METHOD PRIVATE push : BOOL
VAR_INPUT
  pNewCT : POINTER TO FB_ContainerDefGrid;
END_VAR
// checks
// - valid param
IF pNewCT = 0 THEN LogError('push: invalid pointer'); RETURN; END_IF
// - list full
IF _nAttachedCTs >= nUpperIndexCTList THEN  // list overflow no free element for processing
  LogError('Worker processing list full, ignore new CT');
  Abort(iCT:=pNewCT^, sReason:='attach failed - too many attached');  // abort new CT (no release because not yet attached)
  RETURN;
END_IF
// - only one CT allowed
IF _nAttachedCTs > 0 AND NOT _bSupportParallelCT THEN
  LogError(Msg:='another container already attached -> ignore new (set error)');
  Abort(iCT:=pNewCt^, sReason:='attach failed - no parallel support');  // abort new CT
END_IF

// add to list
_nAttachedCTs := _nAttachedCTs + 1;
_pAttachedCTList[_nAttachedCTs] := pNewCT;
MEMSET(destAddr:=ADR(_stAttachedCTData[_nAttachedCTs]), fillByte:=0, n:=SIZEOF(_stAttachedCTData[1]));  // clear additional data
_pNewAttachedHdlData := ADR(_stAttachedCTData[_nAttachedCTs]);   // select handling data for new attached ct 

// apply head
IF _nAttachedCTs = 1 THEN
  // set HEAD
  _pAttachedCt := _pAttachedCTList[nLowerIndexCTList];  
  _bAttached := TRUE;

  // start callback on HEAD
  StartCT(pCtDefGrid:=_pAttachedCt);
END_IF

push := TRUE;
END_METHOD

(*
  Release CT from Worker.
  :return: TRUE if CT was released, FALSE if no CT was registered 
*)
METHOD Release : BOOL
VAR_INPUT
  iCT              : I_CT;                         (*container at triggered event position*)
END_VAR
VAR
  nIdx             : DINT;
  pCT              : POINTER TO FB_ContainerDefGrid;
END_VAR
// remove CT -----------------------------------------------------
// -- get real instance
pCT := getCtInst(iCT:=iCT);
IF pCT = 0 THEN LogError('Release: could not find ct instance'); RETURN; END_IF

// remove and release CT
IF pull(pRemCT:=pCT, nRemIndex=>nIdx) THEN
  LogLvl(Lvl:=E_LogSeverity.Debug, Msg:=F_Concat4('Release CT[', TO_STRING(nIdx), '] ', pCt^.print(0)));
  Release := TRUE;  
END_IF
END_METHOD

(*
  Container will be released from tracker (destroyed) and not available anymore. 
*)
METHOD remove
VAR_INPUT
	(*container at triggered event position*)
	iCT	: I_CT;
END_VAR
SUPER^();

// nothing done
// We keep in internal WorkerList until work is done. CT will be removed from tracker.
END_METHOD

METHOD PRIVATE setName : BOOL
VAR_INPUT
  sName : STRING;
END_VAR
VAR
  nIdx : INT;
  bDone : BOOL;
END_VAR
IF sName = '' THEN
  // generate worker name
  _name := THIS^.InstanceName;
  WHILE NOT bDone DO
    nIdx := FIND(_name, '.');
    IF nIdx = 0 THEN bDone := TRUE; EXIT; 
    ELSE
      _name := RIGHT(_name,LEN(_name)-nIdx);
    END_IF 
  END_WHILE
ELSE
  _name := sName;  
END_IF
END_METHOD

METHOD PROTECTED StartCT
VAR_INPUT
 pCtDefGrid   : POINTER TO FB_ContainerDefGrid;
END_VAR
(* Override specific implementation in child class *)
END_METHOD

METHOD PROTECTED StopCT
VAR_INPUT
 pCtDefGrid   : POINTER TO FB_ContainerDefGrid;
END_VAR
(* Override specific implementation in child class *)
END_METHOD

METHOD  work
VAR
  i : UDINT;
  pCt : POINTER TO FB_ContainerDefGrid;
END_VAR
// set tracking offset
_nTrackOffset := F_MeterToSubPixel(fPosMeter:=fPosition, fResoSubPx:=_fPrintResolution*_fSubPxResolution);  // [pos domain] save position

//Work only with attached container
IF _nAttachedCTs = 0 THEN RETURN; END_IF

IF _pAttachedCt <> 0 AND_THEN _pAttachedCt^.pCT <> 0 THEN _nHeadCtId := _pAttachedCt^.pCT^.iId;
ELSE                                                      _nHeadCtId := 0; END_IF

FOR i:=nLowerIndexCTList TO nLowerIndexCTList + _nAttachedCTs - 1 DO
  pCt := _pAttachedCTList[i];

  // update CT position
  _stAttachedCTData[i].fPosRelToAttach := getPosRelToAttach(iCT:=pCt^);
  
  // release CT (manually)
  IF _bForceRelease THEN
    _bForceRelease := FALSE;
    pCt^.AbortDeformation(sReason:='Manually realease CT', Src:=_pEcSrc^, bHideLog:=FALSE);
    Release(iCT:=pCt^);

  // security release 
  ELSIF _fCtSecurityReleasePos > 0 AND (ABS(_stAttachedCTData[i].fPosRelToAttach) > _fCtSecurityReleasePos) THEN
    pCt^.AbortDeformation(sReason:=F_Concat2('Security released CT Id=', TO_STRING(pCt^.pCT^.iId)), Src:=_pEcSrc^, bHideLog:=FALSE);
    Release(iCT:=pCt^);
  END_IF

END_FOR
END_METHOD

END_FUNCTION_BLOCK

// ---- POUs/Print/DefGrid/FB_WorkerDefGrid_Deformation.TcPOU
FUNCTION_BLOCK FB_WorkerDefGrid_Deformation EXTENDS FB_WorkerDefGrid
VAR_INPUT
END_VAR
VAR_OUTPUT
END_VAR
VAR
  // references
  _iParamMediator : I_ParamMediator;
  
  //Worker specific configuration
  _nPrintUnitWidth            : UDINT;  // default print unit width [px]  
  _nImageWidthPx              : UDINT;  // size of the image (width)
  _nImageDepthPx              : UDINT;  // size of the image (depth)
  
  // -
  _bNewJob                    : BOOL;   // new job started 

  //Deformation status (per attached CT)
  _nDeformationProcPoints     : ARRAY[nLowerIndexCTList..nUpperIndexCTList] OF UDINT;  // available grid points on ct
  _nDeformationProcCols       : ARRAY[nLowerIndexCTList..nUpperIndexCTList] OF UDINT;  // number of already generated grid columns
  _eDeformStep                : ARRAY[nLowerIndexCTList..nUpperIndexCTList] OF E_DeformationStep;   // status deformation of ct
  _bDeformationError          : ARRAY[nLowerIndexCTList..nUpperIndexCTList] OF BOOL;   // status deformation of ct
  _bDeformationBusy           : ARRAY[nLowerIndexCTList..nUpperIndexCTList] OF BOOL;   // status deformation of ct
  _bDeformationDone           : ARRAY[nLowerIndexCTList..nUpperIndexCTList] OF BOOL;   // status deformation of ct
  _nDeformationErrorId        : ARRAY[nLowerIndexCTList..nUpperIndexCTList] OF UDINT;  // status deformation of ct
  _tDeformationExecutionTime  : ARRAY[nLowerIndexCTList..nUpperIndexCTList] OF TIME;   // status deformation of ct
  _bAborted                   : ARRAY[nLowerIndexCTList..nUpperIndexCTList] OF BOOL;   // status deformation of ct

  // ui
  eDeformTypeUi : E_DeformationType;
END_VAR 

VAR PERSISTENT
  _sDeformationGridSettings  : ST_DefGridSettings := (   // grid definition settings
                                  nGridPitchX:=GVL_Deformation.nC_DefaultGridPitch_X,   // this must match the hw config (in fpga)
                                  nGridPitchY:=GVL_Deformation.nC_DefaultGridPitch_Y,   // this must match the hw config (in fpag)
                                  eDeformationType:=E_DeformationType.NoDeformation
                             );
  _fDistToCam                : LREAL := 0.02;   // distance to cam worker 
END_VAR

METHOD PROTECTED  Attach : BOOL
VAR_INPUT
  iCT              : I_CT;                         (*container at triggered event position*)
END_VAR
VAR
  i : UDINT;
  bDeformErr : BOOL;
  eDeformStep : E_DeformationStep;
END_VAR
(*Please do enable externally in PrintModule
IF getCtInst(iCT:=iCT, pCT=>pCt) = 0 THEN    // get specific container
  RETURN;
END_IF

//-- (auto-) enable / disable worker based on mode (do before parent Attach(), is checked inside)
bWorkerEnable := _sDeformationGridSettings.eDeformationType <> E_DeformationType.NoDeformation 
                     AND SEL(pCt^.eCamMode > E_CameraMode.NoCorrection, FALSE, TRUE);
*)

// -- Attach
IF NOT SUPER^.Attach(iCT:=iCT) THEN
  RETURN;
END_IF

// Additional worker checks
IF _pNewAttached = 0 THEN RETURN; END_IF

// - Additional worker checks
bDeformErr := _pNewAttached^.getDeformationStatus(eDStep=>eDeformStep);   // get latest status 
  
// - deformation started? and no deformation error so far
IF bDeformErr OR eDeformStep < E_DeformationStep.cameraStarted THEN
  Release(iCT:=iCT);  // nothing to do anymore

  // - job is valid?
ELSIF _pNewAttached^.pJob = 0 OR NOT _bJobActive THEN
  _pNewAttached^.AbortDeformation(sReason:='No valid job', Src:=_pEcSrc^, bHideLog:=FALSE);
  Release(iCT:=iCT);
  
// - did camera start?  
(*ELSIF eDeformStep < E_DeformationStep.cameraStarted THEN
  _pNewAttached^.AbortDeformation(sReason:='Prio steps did not start', Src:=_pEcSrc^);
  Release(iCT:=iCT);
*)
  
// - OK attach
ELSE
  // checks
  IF eDeformStep < E_DeformationStep.cameraStarted THEN LogWarning('Sub-optimal timing, camera did not yet start'); END_IF
  // start deformation
  _pNewAttached^.StartDeformation(
    sDefGridSettings:=_sDeformationGridSettings, 
    fStartDeformationPos:=getPosRelToAttach(iCT)/_fSubPxResolution   // [px]
  );
  Attach := TRUE;
END_IF
END_METHOD

METHOD InitWorkerDeformation : BOOL
VAR_INPUT
  nPrintUnitWidth : UDINT;
  iDefGridParamMediator : I_ParamMediator;
END_VAR
VAR
  i : UDINT;
END_VAR
IF NOT bInitialized THEN LogError('Base Worker not initialized! call init() before'); RETURN; END_IF
IF iDefGridParamMediator = 0 THEN bInitialized := FALSE; LogError('Invalid parameter, no valid param mediator'); RETURN; END_IF


// worker specific init
_nPrintUnitWidth := nPrintUnitWidth;
_iParamMediator := iDefGridParamMediator;
_bNewJob := FALSE;

FOR i:=nLowerIndexCTList TO nUpperIndexCTList DO
  _nDeformationProcPoints[i]     := 0;
  _nDeformationProcCols[i]       := 0;
  _eDeformStep[i]                := 0;
  _bDeformationError[i]          := 0;
  _bDeformationBusy[i]           := 0;
  _bDeformationDone[i]           := 0;
  _nDeformationErrorId[i]        := 0;
  _tDeformationExecutionTime[i]  := T#0S;
  _bAborted[i]                   := 0;
END_FOR
END_METHOD

METHOD mJobStart
VAR_INPUT
	sJobDef	: CalmarCompPrint.I_JobDefinition;
END_VAR
VAR
  sCamSettings : ST_CameraGridSettings;
END_VAR
// check and init invalid settings
IF _iParamMediator = 0 THEN LogError('no parameter mediator'); RETURN; END_IF
IF _sDeformationGridSettings.nGridPitchX = 0 THEN _sDeformationGridSettings.nGridPitchX:=GVL_Deformation.nC_DefaultGridPitch_X; LogError(F_Concat2('nGridPitchX not configured, set default=', TO_STRING(GVL_Deformation.nC_DefaultGridPitch_X))); END_IF
IF _sDeformationGridSettings.nGridPitchY = 0 THEN _sDeformationGridSettings.nGridPitchY:=GVL_Deformation.nC_DefaultGridPitch_Y; LogError(F_Concat2('nGridPitchY not configured, set default=', TO_STRING(GVL_Deformation.nC_DefaultGridPitch_Y))); END_IF
IF _nPrintUnitWidth = 0 THEN LogError('_nPrintUnitWidth not configured'); END_IF
IF fPosition = 0 THEN LogError('No valid Worker position: set it to WorkerCamera.fCameraToPrintOffset + 0.05; '); END_IF

// configuration
// calculate deformation  settings
// - save image y-offset (centered)
// - save image size
_nImageWidthPx := DINT_TO_UDINT(F_MeterToSubPixel(fPosMeter:=sJobDef.fImageWidth/1000, fResoSubPx:=_fPrintResolution));
_nImageDepthPx := DINT_TO_UDINT(F_MeterToSubPixel(fPosMeter:=sJobDef.fImageDepth/1000, fResoSubPx:=_fPrintResolution));
_sDeformationGridSettings.nGridImageOffsetY := LIMIT(0, ((_nPrintUnitWidth - _nImageWidthPx)) / 2, (_nPrintUnitWidth));  // TODO: if you can get this value from PUC use the other one to have a consistent image shift value 

// - calc grid size and number of points
(*
  Use image width / depth in px divide by GridPitch in X/Y to do a ceil(always next bigger integer).
  +1 -> Because Grid starts at 0 until the calculated numbers we have one point more [0, 1, 2, 3] = 4 points (not 3) 
*)
IF _sDeformationGridSettings.nGridPitchX > 0 AND _sDeformationGridSettings.nGridPitchY > 0 THEN
  _sDeformationGridSettings.nGridSizeX := F_Ceil(val:=UDINT_TO_LREAL(_nImageDepthPx)/_sDeformationGridSettings.nGridPitchX) + 1;
  _sDeformationGridSettings.nGridSizeY := F_Ceil(val:=UDINT_TO_LREAL(_nImageWidthPx + _sDeformationGridSettings.nGridImageOffsetY)/_sDeformationGridSettings.nGridPitchY) + 1;
END_IF
_sDeformationGridSettings.nGridPoints :=  _sDeformationGridSettings.nGridSizeX * _sDeformationGridSettings.nGridSizeY;

sCamSettings := _iParamMediator.sCameraGridSettings;
_sDeformationGridSettings.eDeformationType := sCamSettings.eDeformationType;   // apply deformation mode (for ui)
eDeformTypeUi := _sDeformationGridSettings.eDeformationType;

_bJobActive := TRUE;
END_METHOD

METHOD  mJobStop
VAR_INPUT
	sStatus	: CalmarCompPrint.I_JobStatus;
END_VAR
_bJobActive := FALSE;
END_METHOD

(*
  Release CT from Worker.
  :return: TRUE if CT was released, FALSE if no CT was registered 
*)
METHOD Release : BOOL
VAR_INPUT
  iCT              : I_CT;                         (*container at triggered event position*)
END_VAR
VAR
  i                : DINT;
  Index            : DINT;
  LowerIndex       : DINT := 1;
  pCt              : POINTER TO FB_ContainerDefGrid;
  eStep            : E_DeformationStep;
END_VAR
IF iCT = 0 OR _nAttachedCTs = 0 THEN RETURN; END_IF

// release from deformation module
IF getCtInst(iCT:=iCT, pCT=>pCt) = 0 THEN LogError('Release: could not find ct instance'); RETURN; END_IF
IF _iParamMediator <> 0 THEN
  pCt^.getDeformationStatus(eDStep => estep);
  IF estep >= E_DeformationStep.createdScriptContainer THEN
    pCt^.StopScript(iCT:=iCT);
    //_pParamMediator^.ReleaseDeformationCT(iCT:=iCT);
  END_IF
END_IF

Release := SUPER^.Release(iCT:=iCT);
END_METHOD

PROPERTY sDeformationGridSettings : ST_DefGridSettings
GET
sDeformationGridSettings := _sDeformationGridSettings;
END_GET
END_PROPERTY

METHOD setupPosition
VAR
  sCamSettings : ST_CameraGridSettings;
END_VAR
IF _pAttachedCt <> 0 THEN RETURN; END_IF    // Update only without attached container

sCamSettings := _iParamMediator.sCameraGridSettings;

// set tracking offset
fPosition := sCamSettings.fDetectToCam + _fDistToCam;
END_METHOD

METHOD  work
VAR
  i : UDINT;
  pCT : POINTER TO FB_ContainerDefGrid;
END_VAR
//-----------------------------------------------------------
SUPER^.work();      // Parent implementation

setupPosition();    // Worker position update

// Work only with attached container (additional work to Base class)
FOR i:=nLowerIndexCTList TO nLowerIndexCTList + _nAttachedCTs - 1 DO
  pCt := _pAttachedCTList[i];
 
  // update deformation handler
  pCT^.UpdateDeformation(fPos:=_stAttachedCTData[i].fPosRelToAttach/_fSubPxResolution);  // pos in [px]
  
  // get status
  _bDeformationError[i] := pCt^.getDeformationStatus(eDStep => _eDeformStep[i], 
                            bBusy => _bDeformationBusy[i],
                            bDone => _bDeformationDone[i],
                            nErrorId => _nDeformationErrorId[i], 
                            tExecutionTime => _tDeformationExecutionTime[i],
                            bAborted => _bAborted[i]);
  _nDeformationProcPoints[i] := pCt^.nAvailableGridPoints;
  _nDeformationProcCols[i]   := pCt^.nAvailableGridCols;
     
  // Release container when all points have been processed or error
  IF _bDeformationDone[i] OR _bDeformationError[i] THEN
    // tag CT with error if deformation had an error
    IF _bDeformationError[i] THEN 
      IF NOT _bAborted[i] THEN
        pCt^.AbortDeformation(sReason:=F_Concat2('WorkerDeformation: ', EC_DefGrid.ecDefGrid_DefGridError.Desc), Src:=_pEcSrc^, bHideLog:=FALSE);
      //not needed ELSE
      //  pCt^.setError(ErrDef:=EC_DefGrid.ecDefGrid_DefGridError, Src:=_pEcSrc^);
      END_IF
    END_IF
    LogLvl(Lvl:=E_LogSeverity.Detail, Msg:=F_Concat4('Done with: CamP=',  TO_STRING(pCT^.nRegisteredCameraPoints), ' GridP=', TO_STRING(pCt^.nAvailableGridPoints)));
    Release(pCt^);
  END_IF
  
END_FOR
END_METHOD

END_FUNCTION_BLOCK

// ---- POUs/Print/DefGrid/FB_PrintOverview.TcPOU
FUNCTION_BLOCK FB_PrintOverview
VAR_INPUT
  fX_m,  fY_m   : LREAL;    // max. x/y position [m]
  nX_px, nY_px  : DINT;     // max. x/y pixel in view
  fPxToMRatio   : LREAL;    // 
  iPrintPosition : I_PrintPosition;
END_VAR

VAR
  // helper
  bInit   : BOOL;
  nCtr    : UDINT;
  nNum    : UDINT;
  
  // config
  _pCTM   : POINTER TO FB_CTManagerDefGrid;
  _pWorkerDefGrid : POINTER TO FB_WorkerDefGrid;
  _fPrintResolution : LREAL;      // [dpi]
  _fSubPixelResolution : LREAL;   // sub pixel resolution
  
  // Container view list
  iCT     : I_CT;
  aCTV    : ARRAY[1..iCPr_MAX_CONTAINER] OF FB_ContainerView;
  // Worker view list
  iWorker : I_Worker;
  aWorkerV: ARRAY[1..nC_MAX_WORKER_VIEWS] OF FB_ViewPositionControl;
  aWorkerFb: ARRAY[1..nC_MAX_WORKER_VIEWS] OF POINTER TO FB_WorkerDefGrid;
  
  // motion and position
  bMovingInd : BOOL;
  fSpeed  : LREAL;
  fbBlink : FB_BLINK;
  t : TIME;
  
  // last container debug
  nGridRowStart : UDINT;  // starting grid colum for Grid debug Visu
  nGridColStart : UDINT;  // starting grid colum for Grid debug Visu
  pLastCT : POINTER TO FB_ContainerDefGrid;   // pointer to last created container
  
  // time
  sCurrentDateTime : STRING;
  
  // view control
  bShowCtDetails : BOOL;
END_VAR
VAR CONSTANT
  nC_MAX_WORKER_VIEWS : UINT := 10;
END_VAR

IF NOT checkConfig() THEN RETURN; END_IF    // check config

// -- show CTs -----------------------
nNum := _pCTM^.nCount;
FOR nCtr := 1 TO nNum DO
  // get CT interface from list
  iCT := _pCTM^.getCT(nIdx:=nCtr);
  IF iCT <> 0 THEN
    // set position
    aCTV[nCtr].setPos(x:=iCT.GetPosRel(iTracker:=_pCTM^.iTracker), y:=0);

    // display
    aCTV[nCtr].bHide := FALSE;
    aCTV[nCtr]( iCT:=iCT, 
                iIdx:=UDINT_TO_UINT(iCT.pCT^.nMemIndex), 
                fPxtoMRatio:=fPxToMRatio, 
                fPosToMFactor := 0.0254 / (_fPrintResolution*_fSubPixelResolution), 
                iTracker:=_pCTM^.iTracker);
  END_IF
END_FOR

FOR nCtr := (nNum+1) TO iCPr_MAX_CONTAINER DO
  aCTV[nCtr].iCT := 0;
  aCTV[nCtr].bHide := TRUE;
END_FOR

// -- show Workers -----------------------
iWorker := _pWorkerDefGrid^.Root;
nCtr := 0;
WHILE iWorker <> 0 DO     // walk through worker chain
  nCtr := nCtr + 1;
  aWorkerFb[nCtr] := iWorker.Inst;  // get fb pointer
  aWorkerV[nCtr].bHide := FALSE;
  aWorkerV[nCtr].setPos(x:=aWorkerFb[nCtr]^.nTrackOffset, y:=0);
  iWorker:=iWorker.Next;
END_WHILE
FOR nCtr := (nCtr+1) TO nC_MAX_WORKER_VIEWS DO
  aWorkerV[nCtr].bHide := TRUE;
END_FOR

// -- show positioning -----------------------
fSpeed := iPrintPosition.getSpeed();
IF LrealIsNaN(x:=fSpeed) THEN
  fSpeed := 0;
END_IF
t := LREAL_TO_TIME(1000-fSpeed*900);
fbBlink(bI_Enable:=SEL(fSpeed > 0, FALSE, TRUE), tI_Time:=t, bO_Out=>bMovingInd);

// -- last container debug detail ------------
IF _pCTM^.nCount > 0 THEN
  iCT := _pCTM^.getCT(1);
  IF iCT <> 0 THEN  pLastCT := _pCTM^.GetContainerInstance(iCT:=iCT); END_IF
END_IF

// -- current time ---------------------------
sCurrentDateTime := F_TimeGetDateTime();

METHOD checkConfig : BOOL
VAR_INPUT
END_VAR
VAR_INST
  _fX_m, _fY_m   : LREAL;
  _nX_px, _nY_px : DINT; 
END_VAR
VAR
  bOK : BOOL;
END_VAR
IF NOT bInit THEN RETURN; END_IF
IF iPrintPosition = 0 THEN RETURN; END_IF

_fPrintResolution := iPrintPosition.fPrintResolution;
_fSubPixelResolution := iPrintPosition.fSubPxResolution;

// changed settings
IF _fX_m <> fX_m OR
          _fY_m <> fY_m OR
          _nX_px <> nX_px OR
          _nY_px <> nY_px THEN
  // save new config
   _fX_m := fX_m;
   _fY_m := fY_m;
   _nX_px := nX_px;
   _nY_px := nY_px;
   config();
END_IF

checkConfig := TRUE;
END_METHOD

METHOD PRIVATE config
VAR_INPUT
END_VAR
// NOTE: some config values are given only here (internally)
FOR nCtr := 1 TO iCPr_MAX_CONTAINER DO
  aCTV[nCtr].init(
    nXPosMin:=0,
    nXPosMax:= F_MeterToSubPixel(fPosMeter := fX_m, fResoSubPx := _fPrintResolution * _fSubPixelResolution),
    nYPosMin:=0,
    nYPosMax:=F_MeterToSubPixel(fPosMeter := fY_m, fResoSubPx := _fPrintResolution * _fSubPixelResolution),
    bXFlip:=TRUE,
    bYFlip:=FALSE,
    nXMinPx:=0,
    nXMaxPx:=nX_px,
    nYMinPx:=0,
    nYMaxPx:=nY_px,
  );
  aCTV[nCtr].setPos(x:=0, y:=0);
END_FOR
FOR nCtr := 1 TO nC_MAX_WORKER_VIEWS DO
  aWorkerV[nCtr].init(
    nXPosMin:=0,
    nXPosMax:= F_MeterToSubPixel(fPosMeter := fX_m, fResoSubPx := _fPrintResolution * _fSubPixelResolution),
    nYPosMin:=0,
    nYPosMax:=F_MeterToSubPixel(fPosMeter := fY_m, fResoSubPx := _fPrintResolution * _fSubPixelResolution),
    bXFlip:=TRUE,
    bYFlip:=FALSE,
    nXMinPx:=0,
    nXMaxPx:=nX_px,
    nYMinPx:=0,
    nYMaxPx:=nY_px,
  );
  aWorkerV[nCtr].setPos(x:=0, y:=0);
END_FOR

bInit := TRUE;
END_METHOD

METHOD init : BOOL
VAR_INPUT
  pCTM  : POINTER TO FB_CTManager;
  pWorkerDefGrid : POINTER TO FB_WorkerDefGrid;
END_VAR
IF pCTM = 0 OR pWorkerDefGrid = 0 THEN RETURN; END_IF

_pCTM := pCTM;
_pWorkerDefGrid := pWorkerDefGrid;

bInit := TRUE;
END_METHOD

END_FUNCTION_BLOCK

// ---- POUs/Print/DefGrid/FB_PrintPositionDmax.TcPOU
FUNCTION_BLOCK FB_PrintPositionDmax EXTENDS FB_BasePrint IMPLEMENTS I_PrintPosition, I_Sim
VAR_INPUT
  IlEncoderPulse      AT%I* : UDINT;                // Encoder counter intput
  IbEncoderWcState    AT%I* : BOOL;                 // Encoder EL5101 WcState
END_VAR
// ----------------------------------
// configuration
VAR
  // configuration (init)
  _fPrintResolution         : LREAL := 600;         // print(head) resolution in [dpi]
  _fSubPxResolution         : LREAL := 32;          // SubPixel resolution [SubPx], resolution factor (fI_PrintResolution*fI_SubPxResolution=>Output resolution)
  _fTaskCycleTime           : LREAL := 0.002;       // Task cycle time in [s]
  
  _fSpeedMpMin              : LREAL;                // speed in [m/min]
  
  // Debug
  // Machine simulation mode
  nSimMode : UINT := 0;   // 0=standard sim PosMaster, 1=ramp up/down 
  fSimSpeed : LREAL := 0.1;   // [m/s]
  bCmdStartPos, bCmdStopPos : BOOL;                 // test command to start/stop simulated the machine
END_VAR
VAR PERSISTENT
  // config - values changable during runtime (recipe, visu, property)
  // - encoder settings 
  _fEncoderResolution       : LREAL := 2.00475;     // Encoder resolution
  // - speed compensation
  _bEnSpeedComp             : BOOL  := FALSE;
  _fSpeedCompFactor         : LREAL := 0.0;         // TODO: define value
  _fSpeedCompRefSpeed       : LREAL := 0.0;         // TODO: define value
END_VAR

// ---------------------------------
// internal variables
VAR
  // fb inst
  fbPositionMaster          : FB_PositionMaster;

  // internal vars
  _bMoving                  : BOOL;
  
  _bStarted                 : BOOL;
  fEncoderReso              : LREAL;                // used encoder resolution (config + speedcomp)
  rTrigMoving               : R_TRIG;
  // simulation
  _bSim                     : BOOL;
  rfTrig_Sim                : RF_TRIG;
END_VAR


// set internal used resolution
fEncoderReso := _fEncoderResolution;  

// compensate resolution (if enabled)
IF _bEnSpeedComp THEN
  fEncoderReso := F_EncoderSpeedComp(   
    fMasterSpeed:=fbPositionMaster.fMasterSpeed,
    fResolution:=_fEncoderResolution,
    fSpeedCompFactor:=_fSpeedCompFactor,
    fSpeedCompRefSpeed:=_fSpeedCompRefSpeed
  );
END_IF

// calc position / speed
fbPositionMaster(fResolutionInput:=fEncoderReso, lPosReference:=IlEncoderPulse);

// position status
_bMoving := ABS(fbPositionMaster.fMasterSpeed) >= fbPositionMaster.fMinSpeed; 
_fSpeedMpMin := fbPositionMaster.fMasterSpeed * 60;
rTrigMoving(CLK:=bMoving);   // create started trigger output
_bStarted := rTrigMoving.Q OR fbPositionMaster.bSyncReq;

// simulation
simulation();

(*
  Position is moving.
*)
PROPERTY bMoving : BOOL
GET
bMoving := _bMoving;
END_GET
END_PROPERTY

{attribute 'monitoring' := 'call'}
(*Simulation is enabled set/get*)
PROPERTY bSimEnable : BOOL
GET
bSimEnable := _bSim;
END_GET
SET
_bSim := bSimEnable;
END_SET
END_PROPERTY

(*
  Started moving event.
*)
PROPERTY bStarted : BOOL
GET
bStarted := _bStarted;
END_GET
END_PROPERTY

(*
  Read / Write Encoder resolution.
*)
PROPERTY fEnoderResolution : LREAL
GET
fEnoderResolution := _fEncoderResolution;
END_GET
SET
_fEncoderResolution := fEnoderResolution;
END_SET
END_PROPERTY

(*
  print(head) resolution in [dpi]
*)
PROPERTY fPrintResolution : LREAL
GET
fPrintResolution := _fPrintResolution;
END_GET
END_PROPERTY

(*
   SubPixel resolution [SubPx]
*)
PROPERTY fSubPxResolution : LREAL
GET
fSubPxResolution := _fSubPxResolution;
END_GET
END_PROPERTY

(*
  Get current "default" position.
  [SubPx] as return value and [um] as output
  :return: position in [SubPx] resolution
*)
METHOD getPosition : DINT
VAR_OUTPUT
  nPosition_px       : DINT;                 // Master position in [px]
  fPosition_um       : LREAL;                // Master position in [um]
END_VAR
getPosition := fbPositionMaster.lMasterPosition;
nPosition_px := fbPositionMaster.lMasterPosition / LREAL_TO_DINT(_fSubPxResolution);
fPosition_um := fbPositionMaster.fMasterPosition;
END_METHOD

(*
  Get "default" speed [m/s].
  :returns: current speed in [m/s]
*)
METHOD getSpeed : LREAL
VAR_OUTPUT
  fSpeedMpMin : LREAL;  // speed in [m/min]
END_VAR
getSpeed    := fbPositionMaster.fMasterSpeed;
fSpeedMpMin := fbPositionMaster.fMasterSpeed*60;
END_METHOD

METHOD Init : BOOL
VAR_INPUT
  fPrintResolution    : LREAL := 600;         // print(head) resolution in [dpi]
  fSubPxResolution    : LREAL := 32;          // SubPixel resolution [SubPx], resolution factor (fI_PrintResolution*fI_SubPxResolution=>Output resolution)
  fTaskCycleTime      : LREAL;                // Task cycle time in [s]
END_VAR
// store config
_fPrintResolution := fPrintResolution;
_fSubPxResolution := fSubPxResolution;
_fTaskCycleTime   := fTaskCycleTime;

// init fbs
// - position master
fbPositionMaster.init(
  fI_PrintResolution:=fPrintResolution, 
  fI_SubPxResolution:=fSubPxResolution, 
  fI_TaskCycleTime:=fTaskCycleTime, 
  bI_HWEncoder:=FALSE
);
END_METHOD

METHOD reset
VAR_INPUT
END_VAR
// reset positioning system
fbPositionMaster.reset();
END_METHOD

METHOD simulation
VAR_INST
  rf_Start, rf_Stop : RF_TRIG;
  fSetSpeed : LREAL;          // [m/s] current sim set speed
  fRampUpTime : LREAL := 2;   // [s] to ramp up/down machine
END_VAR
rfTrig_Sim(CLK:=_bSim);
IF rfTrig_Sim.RT THEN fbPositionMaster.bSim:=TRUE; END_IF
IF rfTrig_Sim.FT THEN fbPositionMaster.bSim:=FALSE; END_IF
fbPositionMaster.fSimSpeed := fSimSpeed;


rf_Start(CLK:=bCmdStartPos);
rf_Stop(CLK:=bCmdStopPos);

IF    nSimMode = 0 THEN
  ; // just use running position with sim speed in PositionMaster

ELSIF nSimMode = 1 THEN
  IF fRampUpTime = 0 THEN RETURN; END_IF
  IF rf_Start.RT THEN fSetSpeed := 0; END_IF  
  // starting
  IF bCmdStartPos THEN
    fSetSpeed := fSetSpeed + (fSimSpeed/fRampUpTime)*_fTaskCycleTime;
    IF fSetSpeed >= fSimSpeed THEN bCmdStartPos:=FALSE; fSetSpeed := fSimSpeed; END_IF
  END_IF
  // stopping
  IF bCmdStopPos THEN
    fSetSpeed := fSetSpeed - (fSimSpeed/fRampUpTime)*_fTaskCycleTime;
    IF fSetSpeed <= 0 THEN bCmdStartPos:=FALSE; fSetSpeed := 0; END_IF
  END_IF
  
ELSIF nSimMode = 2 THEN
  // sim encoder signal (if not fbPositionMaster is used)
  IF _bSim THEN // sim encoder pulse
    IlEncoderPulse := TO_UDINT(TO_DINT(IlEncoderPulse) + TO_DINT(((fbPositionMaster.fSimSpeed * _fTaskCycleTime)*1_000_000)/SEL(_fEncoderResolution=0, _fEncoderResolution, 1)));
  END_IF
  
END_IF
END_METHOD

END_FUNCTION_BLOCK

// ---- POUs/Print/DefGrid/F_EncoderSpeedComp.TcPOU
(*
  Encoder speed compensation.
  
  NOTE: Calculation can be disabled by setting fSpeedCompFactor=0
  :return: compensated encoder resolution
*)
FUNCTION F_EncoderSpeedComp : LREAL
VAR_INPUT
  (* live value *)
  fMasterSpeed                  : LREAL;		        (*Current Speed in [m/s]*)
  (* configuration *)
  fResolution                   : LREAL := 0.0;     (*default encoder resolution*)
  fSpeedCompFactor              : LREAL := 0.0;     (*TODO: define value*)
  fSpeedCompRefSpeed            : LREAL := 0.0;     (*TODO: define value*)
END_VAR
VAR
  fL_Compensation               : LREAL := 0.0;
END_VAR

IF (fSpeedCompFactor <> 0) AND (fMasterSpeed <> 0) THEN
  
  (*Calculate compensation*)
  fL_Compensation := (fMasterSpeed - fSpeedCompRefSpeed) * fSpeedCompFactor;
  fL_Compensation := DINT_TO_LREAL(FC_LREAL_TO_DINT(fL_Compensation * 10_000)) / 10_000;	(*Rounding to prevent small changes oscillation*)
  
  F_EncoderSpeedComp := fResolution * (1 + fL_Compensation);
ELSE
  
  (*return input resolution*)
  F_EncoderSpeedComp := fResolution;
END_IF;

END_FUNCTION

// ---- POUs/Print/DefGrid/FB_ProdManager_DMAX.TcPOU
(*
  Managing a production on a DigiRound machine.
*)
FUNCTION_BLOCK FB_ProdManager_DMAX EXTENDS FB_BasePrint IMPLEMENTS I_PrintStatusClient, I_ProdManager
VAR
 //references
  _pPU                : POINTER TO FB_PU;               (*PU reference*)
  
  //settings
  _defaultPrintData   : ST_PRINT_SETTING;               (*default PDI data if no CT present*)
  _isVarData          : BOOL; 

  //status
  bPmActive           : BOOL;                           (*a production is active*)
  rfTrig_PmActive     : RF_TRIG;
  lastCreatedCT       : I_CT;                           (*last created container*)
  sActiveJobInfo      : T_MaxString;                    (*current job information string*)
  nScrap              : UDINT;
  nProduced           : UDINT;
  nToProduce          : UDINT;

  (*lists*)
  (*--job trace list*)
  _currJobId          : STRING;                         (*id of current started job*)

  (*internals*)
  _pEcSrc : POINTER TO T_ErrSrc;                                    (*error source definition*)

END_VAR
VAR CONSTANT
  lNUM_LIST_SIZE        : DINT := iCPr_MAX_CONTAINER;   (*number of max. list elements*)
  // other logs
  aC_Dbg_NotReject      : STRING := 'could not rejectNext CT';
  aC_Dbg_InvPtrCT       : STRING := 'invalid pO_ContainerHead';
  aC_Dbg_InvPtrJob      : STRING := 'invalid Job pointer';
  aC_Ddb_GetNext        : STRING := 'getNext from: ';  
END_VAR

IF NOT bInitialized THEN RETURN; END_IF  // ignore

rfTrig_PmActive(CLK:=bPmActive);

(*
  Job was stopped. 
  :return: TRUE if some elements were aborted in machine.
*)
METHOD PRIVATE abortJob : BOOL
VAR
END_VAR
// a job stopped.

// NOTE: not implemented
END_METHOD

PROPERTY bReady : BOOL
GET
bReady := bPmActive;
END_GET
END_PROPERTY

PROPERTY bStarted : BOOL
GET
bStarted := rfTrig_PmActive.RT;
END_GET
END_PROPERTY

PROPERTY bStopped : BOOL
GET
bStopped := rfTrig_PmActive.FT;
END_GET
END_PROPERTY

(*
Create/Build a new container (CT) with next page to be printed.
*)
METHOD CT_Create : BOOL
VAR_INPUT
  sCT            : I_CT;                  // container to produce
END_VAR
VAR 
  _created       : BOOL := FALSE;
  sPage          : ST_PrintPageDef;
END_VAR
// prepare & checks
lastCreatedCT := 0;                      // invalidate last created
IF NOT bInitialized THEN RETURN; END_IF
IF sCT = 0 THEN LogError(aC_Dbg_InvPtrCT); RETURN; END_IF

(* getNext CT *)
IF getNext(sCT := sCT) THEN
  
  // define printer output
  sPage := sCT.sPageDef;
  IF    sPage.lType = EN_PrintPageType.maintenance THEN // - maintenance
    sCT.pCT^.lPrOutput := EN_PrinterOutput.trash;     // -> eject trash
  ELSIF sPage.lType = EN_PrintPageType.production OR   // - production
        sPage.lSrc = EN_PrintPageSrc.overprod OR       // - over-production
        sPage.lType = EN_PrintPageType.separator THEN  // - separator 
    sCT.pCT^.lPrOutput := EN_PrinterOutput.prod;      // -> production output
  ELSE                                                // - rest
    sCT.pCT^.lPrOutput := EN_PrinterOutput.trash;     // -> eject trash
  END_IF

  lastCreatedCT := sCT;                // successfully produced a CT, store last created CT (necessary for async access within this cycle)
  sCT.pCT^.bCreated := TRUE;
  _created := TRUE;
ELSE
  sCT.setError(EC_Print.ecPMInvGetNext, Src:=_pEcSrc^);   // getNext error
END_IF

(* logging *)
LogLvl(Lvl:=E_LogSeverity.Debug, Msg:=CONCAT('create CT: ', sCT.print(0)));

(*return value*)
CT_Create := _created;
END_METHOD

METHOD CT_Finish : BOOL
VAR_INPUT
  sCT            : I_CT;               // container to produce
  bSuccess       : BOOL;               // printed OK?
END_VAR
VAR
  bErr           : BOOL;
END_VAR
(* checks *)
IF NOT bInitialized THEN RETURN; END_IF                             // exit if no production is active
IF sCT = 0 THEN LogError(aC_Dbg_InvPtrCT); RETURN; END_IF  // log invalid pointer 

// tag machine errors on CT
IF sCT.pCT^.bValid AND NOT bSuccess THEN  
    sCT.setError(EC_Print.ecPMCTMachineErr, Src:=_pEcSrc^);            // tag CT with: error from machine 
END_IF

// report page done to PU
IF NOT sCT.pCT^.bReported AND sCT.pJob <> 0 THEN
  IF _pPU^.endPage(sCT:=sCT, bSuccess:=bSuccess) THEN
    ;
  ELSE
    sCT.setError(EC_Print.ecPMInvSet, Src:=_pEcSrc^);
  END_IF
END_IF

(* logging *)
IF bSuccess THEN
  LogLvl(Lvl:=E_LogSeverity.Detail, Msg:=CONCAT('successCT: ', sCT.print(0)));
ELSE
  LogLvl(Lvl:=E_LogSeverity.Detail, Msg:=CONCAT('eject  CT: ', sCT.print(0)));  
END_IF

(* return value *)
CT_Finish := TRUE;
END_METHOD

(*
  Finalize/Produce a CT. Now we shouldhave all necessary information for configuring the CT.
*)
METHOD CT_Produce : BOOL
VAR_INPUT
  sCT                 : I_CT;               // container to produce
END_VAR
VAR
  _produced           : BOOL := FALSE;
  sPage               : ST_PrintPageDef;
  bPresent            : BOOL;
END_VAR
(* parameter checks *)
IF NOT bInitialized THEN RETURN; END_IF
IF sCT = 0 THEN LogError(aC_Dbg_InvPtrCT); RETURN; END_IF

sCT.pCT^.bValid           := TRUE;                (* we have all data - CT is valid configured*)

// reject page if no container present or overproduction
sPage := sCT.sPageDef;
bPresent := sCT.pCT^.bProductPresent;
IF NOT bPresent AND sPage.lSrc <> EN_PrintPageSrc.overprod  THEN
  (*   add it to rejected queue (high prio reproduction), we will try to produce this CT in next cycle*)
  IF NOT _pPU^.rejPage(sCT:=sCT) THEN
    LogLvl(Lvl:=E_LogSeverity.Info, aC_Dbg_NotReject);
  END_IF
END_IF

(* logging *)
IF bPresent THEN LogLvl(Lvl:=E_LogSeverity.Detail,  Msg:=CONCAT('produceCT: ', sCT.print(0)));
            ELSE LogLvl(Lvl:=E_LogSeverity.Debug,   Msg:=CONCAT('produceCT: ', sCT.print(0))); END_IF

(* return value*)
CT_Produce := _produced;
END_METHOD

PROPERTY defaultPrData : ST_PRINT_SETTING
GET
defaultPrData := _defaultPrintData;
END_GET
END_PROPERTY

METHOD PRIVATE dynAddPage : BOOL
VAR_INPUT
  lType     : EN_PrintPageType; 
  lPageNr   : UDINT;
END_VAR
IF _pPU = 0 THEN F_Report_Error(ErrType:=EN_REPORT_ERROR_TYPE.Report_Error_0Pointer); RETURN; END_IF
IF lType <> EN_PrintPageType.maintenance THEN
  LogError('dynAddPage: only supports maintenance pages'); 
END_IF

_pPU^.addPage(
  lPageType:=EN_PrintPageType.maintenance,
  lPageSrc:=EN_PrintPageSrc.Sample,
  lPageNr:=1
);
END_METHOD

(*
  get next page to be printed.
  :return:    TRUE if success.
*)
METHOD PRIVATE getNext : BOOL               (*get next image to be printed*)
VAR_INPUT
  sCT               : I_CT;                 (*container handle*)
END_VAR
VAR
  bErr              : BOOL;
  lRemainingPages   : UDINT;
END_VAR
VAR_INST
  rTrig_PreStop     : R_TRIG;
END_VAR
IF NOT bInitialized THEN RETURN; END_IF                    (* Exit if no production is active*)

// ask pu for a next page
bErr := NOT _pPU^.getPage(sCT:=sCT, lPagesLeft=>lRemainingPages);

getNext := NOT bErr;
END_METHOD

METHOD init : BOOL
VAR_INPUT
  pPU     : POINTER TO FB_PU;
  // machine specific
END_VAR
// parameter checks
IF pPU = 0 THEN
  F_Report_Error(ErrType:=EN_REPORT_ERROR_TYPE.Report_Error_0Pointer);
  RETURN;
END_IF

// register external references
_pPU := pPU;

// init error source
_pEcSrc := ErrorCodes.fbErrCodeMngr.registerErrSource(
  nLocId:=0, 
  aInstPath:=InstanceName, 
  aLocDescr:='PrintManager DMAX'
);
IF _pEcSrc = 0 THEN LogError('could not register error source'); END_IF

//reset setates
bPmActive := FALSE;
lastCreatedCT := 0;

bInitialized := TRUE;
END_METHOD

METHOD JobFinished : BOOL
VAR_INPUT
  aSeparatorId   : STRING;
END_VAR
// Job Handling -----------------------

// NOTE: nothing implemented for now
END_METHOD

PROPERTY lastCreated : I_CT
GET
lastCreated := lastCreatedCT;
END_GET
END_PROPERTY

METHOD mJobPause
END_METHOD

METHOD mJobStart
VAR_INPUT
	sJobDef	: I_JobDefinition;
END_VAR
VAR
  n1,n2,n3 : UDINT;
END_VAR
IF NOT bInitialized THEN RETURN; END_IF
IF sJobDef = 0 THEN RETURN; END_IF

// start job 
LogLvl(lvl:=E_LogSeverity.Detail, Msg:=F_Concat5('PM start job: ', sJobDef.aJobId, ' (', sJobDef.aJobName, ')'));

// setup PrintManager with new job
_currJobId := sJobDef.aJobId;
_isVarData := sJobDef.isVarData();

// -- init last created
lastCreatedCT := 0;

// -- init defaultPrintData (TODO: not sure why we really need this)
MEMSET(ADR(_defaultPrintData), 0, SIZEOF(_defaultPrintData));   // reset default data

// -- add pre-production pages (product specific) -> maintenance pages
(*FOR lCt := 1 TO lStartEject DO 
  dynAddPage(lType:=EN_PrintPageType.maintenance, 1);
END_FOR*)

bPmActive := TRUE;
sActiveJobInfo := F_Concat7(
  F_Concat3('Name:      ', sjobdef.aJobName, '$n'),
  F_Concat3('JobId:     ', sjobdef.aJobId, '$n'),
  F_Concat3('FlowId:    ', sjobdef.aFlowId, '$n'),
  F_Concat3('Substrate: ', sjobdef.aSubstrateName, '$n'),
  F_Concat3('Descr:     ', sjobdef.aJobDescription, '$n'),
  F_Concat4('Width:     ', TO_STRING(sjobdef.fImageWidth), ' [mm]', '$n'),
  F_Concat4('Depth:     ', TO_STRING(sjobdef.fImageDepth), ' [mm]', '$n')
);

sJobDef.getJobPageNbrs(nProdPages=>n1, nMaintPages=>n2, nPrePrPages=>n3);
nToProduce := n1+n2;
END_METHOD

METHOD mJobStop
VAR_INPUT
	sStatus	: I_JobStatus;
END_VAR
IF NOT bInitialized THEN RETURN; END_IF

(*Stop job*)
LogLvl(lvl:=E_LogSeverity.Detail, Msg:=
  F_Concat7(
    'PM stop job P(',
    TO_STRING(sStatus.iJobProgress.lProductionCount), ') M(',
    TO_STRING(sStatus.iJobProgress.lMaintenanceCount), ') S(',
    TO_STRING(sStatus.iJobProgress.lScrapCount), ')'
  )
);

abortJob();

bPmActive := FALSE;
sActiveJobInfo := 'No job active';
nProduced := nScrap := 0;
lastCreatedCT := 0;
END_METHOD

METHOD mProduced
VAR_INPUT
	(* current progress*)
	sProgress	: I_JobProgress;
END_VAR
IF NOT bInitialized THEN RETURN; END_IF

nProduced  := sProgress.lProductionCount + sProgress.lMaintenanceCount;
nScrap     := sProgress.lScrapCount;
END_METHOD

END_FUNCTION_BLOCK

// ---- POUs/Print/DefGrid/FB_PythonInterface.TcPOU
FUNCTION_BLOCK FB_PythonInterface EXTENDS T_NamedBase
VAR
  // interface paths (config)
  sPythonInterfacePath : STRING(255); //e.g. 'PRG_x.fb_PythonInterface'
  sPythonContainerPath : STRING(255); //e.g. 'PRG_x.fb_ContainerManager.sL_Containers[%id%].fb_ImageDeformation'
  sPythonScriptPath    : STRING(255);

	bPythonHeartbeat : BOOL;      // <- script is toggling this value as long as it's alive (for plc watchdog of script)
	nPythonPID : UDINT := 0;      // <- python process id (evaluated and given by external script)
  nPythonNewJob : DINT;         // -> new job indication to script
  bPythonNewJobDone : BOOL;     // <- new job registered/done by script

	nContainerToRegister : DINT := -1; // <- triggers a new container creation, except if < 0
  nContainerToRegister_mem : DINT := -1;
	nContainerToDelete : DINT := -1;   // <- triggers a new container deletion, except if < 0
  nContainerToDelete_mem : DINT := -1;
  
  // job definition
  aPythonJobName : T_MaxString; // -> new job name
  aPythonJobGuid : T_MaxString; // -> new job GUID
  //Job settings all in [px]
  nPythonImageOffsetY : UDINT := 0;     // [px]  y offset from 0 to source image
  nPythonImageWidth : UDINT := 1000;    // [px]  source image width (depth)
  nPythonImageHeight  : UDINT := 1000;  // [px]  source image height (width)
  //Grid settings
  nPythonGridPitchX  : UDINT := 100;    // [px]
  nPythonGridPitchY  : UDINT := 100;    // [px]
  nPythonGridSizeX   : UDINT := 0;      // (not yet used) number of grid columns
  nPythonGridSizeY   : UDINT := 0;      // (not yet used) number of grid rows
  //Cam specific settings
  nPythonCamFrameWidth  : UDINT := 200; // [px]
  
  nState : UDINT;
  fbStateTimer : TON;
  fBScriptLauncher : FB_ScriptLauncher;
  _bEnable : BOOL;
  _bKeepAlive : BOOL := TRUE; // keep script alive (restart after crash/close)
  _nStarts : UDINT;   // number of script start attempts
  _nErrCtr : UDINT;   // script error state counter
  _bBusy : BOOL;
  _nErrId : UDINT;
  _bJobStartRequest: BOOL;
  _bJobStopRequest: BOOL;
  _bResetError : BOOL;    // reset state machine error 
  _nJobIdCtr : DINT;
 
	// Python script heartbeat
	fbWatchdog : TOF;
	tWatchdogPeriod : TIME := T#1S;
	fbHeartbeat1 : R_TRIG;
	fbHeartbeat2 : F_TRIG;
	bScriptAlive : BOOL;

END_VAR

VAR CONSTANT
  cStateIdle      : UDINT := 0;
  cStateStartup   : UDINT := 10;
  cStartScript    : UDINT := 20;
  cStateRunning   : UDINT := 30;
  cStateJobActive : UDINT := 40;
  cStateError     : UDINT := 50;
  cStateStop      : UDINT := 60;
  cStateStopping  : UDINT := 70;
  
  cMaxStartAttempts : UDINT := 5;
END_VAR

InterfaceStateMachine();

// reset Container commands, so we suer have a change event on index
IF nContainerToRegister >= 0 AND nContainerToRegister_mem >= 0 THEN nContainerToRegister := -1; END_IF
IF nContainerToDelete >= 0 AND nContainerToDelete_mem >= 0 THEN nContainerToDelete := -1; END_IF
nContainerToRegister_mem := nContainerToRegister;
nContainerToDelete_mem := nContainerToDelete;

fbHeartbeat1(CLK := bPythonHeartbeat);
fbHeartbeat2(CLK := bPythonHeartbeat);
fbWatchdog(IN := fbHeartbeat1.Q OR fbHeartbeat2.Q, PT:=tWatchdogPeriod);
bScriptAlive := fbWatchdog.Q AND nPythonPID <> 0;

METHOD ackError
VAR_INPUT
END_VAR
_bResetError := TRUE;
END_METHOD

{attribute 'monitoring':='call'}
PROPERTY bBusy : BOOL
GET
bBusy := _bBusy;
END_GET
END_PROPERTY

PROPERTY bEnable : BOOL
GET
bEnable := _bEnable;
END_GET
SET
_bEnable := bEnable;
END_SET
END_PROPERTY

{attribute 'monitoring':='call'}
PROPERTY bError : BOOL
GET
IF nState = cStateError THEN bError := TRUE; END_IF;
END_GET
END_PROPERTY

{attribute 'monitoring':='call'}
PROPERTY bJobActive : BOOL
GET
IF nState = cStateJobActive THEN bJobActive := TRUE; END_IF;
END_GET
END_PROPERTY

{attribute 'monitoring':='call'}
PROPERTY bRunning : BOOL
GET
IF nState = cStateRunning THEN bRunning := TRUE; END_IF;
END_GET
END_PROPERTY

METHOD Init : BOOL
VAR_INPUT
  sCTManagerPath : T_MaxString;  // ct manager path (plc variable instance path)
  sScriptPath    : T_MaxString;  // path to python script base folder, e.g. C:\Work\script
END_VAR
sPythonInterfacePath := THIS^.InstanceName;
sPythonContainerPath := sCTManagerPath;
sPythonScriptPath    := sScriptPath;

// init launcher
fBScriptLauncher.Init(sPythonScriptPath);

// some variable init
aPythonJobName := 'JobNameUnknown';
aPythonJobGuid := 'aaaaaaaa-bbbb-cccc-dddd-eeeeeeeeeeee';

//Launch init procedure
fbStateTimer(PT:=T#5S);
nState := cStateIdle;
END_METHOD

ACTION InterfaceStateMachine:

CASE(nState) OF
  // Idle
  cStateIdle  :
    _bJobStartRequest:=FALSE;
    _bJobStopRequest:=FALSE;
    _bResetError := FALSE;
    IF bEnable THEN
      nState := cStateStartup;
    END_IF  

  //Startup
  cStateStartup   :
    fbStateTimer(IN:=TRUE);         // start timeout
    _bBusy := TRUE;

    IF fbStateTimer.Q THEN
      fbStateTimer(IN:=FALSE);
      _nStarts := _nStarts + 1;
      IF bScriptAlive THEN
        nState := cStateRunning;    // is already running
      ELSE  
        RunPythonScript();          // start script
        nState := cStartScript;
			END_IF
		END_IF
  
  //Start Python script and wait until it starts
  cStartScript    :
    fbStateTimer(IN:=TRUE);
    _bBusy := TRUE;

    IF NOT fBScriptLauncher.bBusy AND bScriptAlive THEN 
      IF fBScriptLauncher.bError THEN //Launch error
        LogError(F_Concat2('Script start error=', TO_STRING(fBScriptLauncher.nErrId)));
        nState := cStateError;
      ELSE //Launch done and heartbeat ok
        nState := cStateRunning;
        fbStateTimer(IN:=FALSE);
			END_IF
    ELSIF fbStateTimer.Q THEN //Timeout error (could not start)
      IF fBScriptLauncher.bError THEN //Launch error
        ///LogError(F_Concat2('Script start error=', TO_STRING(fBScriptLauncher.nErrId)));
        LogError(F_Concat2('Script start error=', F_GetAdsErrStr(fBScriptLauncher.nErrId)));
      ELSE
        LogError('Script start error');
      END_IF
      nState := cStateError;
		END_IF
 
  //Script running with correct watchdog feedback
  cStateRunning   : 
    fbStateTimer(IN:=_bJobStartRequest);
    _bBusy := _bJobStartRequest;
    _bJobStopRequest := FALSE;
    _nStarts := 0;
    
    IF _bJobStartRequest AND bPythonNewJobDone THEN
      _bJobStartRequest:=FALSE;
      bPythonNewJobDone := FALSE; 
      fbStateTimer(IN:=FALSE);  
      nState := cStateJobActive;
    ELSIF NOT bScriptAlive THEN //Watchdog error
      LogError('Script watchdog error');
      nState := cStateError;
    ELSIF fbStateTimer.Q THEN //Job timeout error
      LogError('Script new job done error');
      nState := cStateError;
    ELSIF NOT bEnable THEN
      nState := cStateStop;
		END_IF
  
  //JobStarted
  cStateJobActive :
    fbStateTimer(IN:=_bJobStopRequest);
    _bBusy := _bJobStopRequest;
    
    IF _bJobStopRequest THEN
      nPythonNewJob := 0;
    END_IF;  
    
    IF _bJobStopRequest THEN
      _bJobStopRequest:=FALSE;
      fbStateTimer(IN:=FALSE);  
      nState := cStateRunning;
    ELSIF NOT bScriptAlive THEN //Watchdog error
      LogError('Script watchdog error');
      nState := cStateError;
    ELSIF fbStateTimer.Q THEN //Job timeout error
      LogError('Script new job done error');
      nState := cStateError;
    ELSIF NOT bEnable THEN
      nState := cStateStop;
		END_IF
  
  //Error  
  cStateError     :
    fbStateTimer(IN:=FALSE);  
    _bJobStartRequest:=FALSE;
    _bJobStopRequest:=FALSE;
    // reset error 
    IF _bResetError THEN
      _nStarts := 0;          // exit error 
      _nErrCtr := _nErrCtr + 1;
      nState := cStateStop ;
    ELSIF NOT bEnable THEN
      nState := cStateStop ;  // just stop
    ELSIF (_bKeepAlive AND _nStarts <= cMaxStartAttempts)  THEN
      _nErrCtr := _nErrCtr + 1;   // retry 
      nState := cStateStop ;
		END_IF
    
  //Stop 
  cStateStop  :
    StopPythonScript();
    nState := cStateStopping;

  // Stopping
  cStateStopping  :
    IF NOT fBScriptLauncher.bBusy THEN 
      IF fBScriptLauncher.bError THEN //Launch error
        LogError(F_Concat2('Script stop errror:', TO_STRING(fBScriptLauncher.nErrId)));
			END_IF
      nState := cStateIdle;
    END_IF

END_CASE
END_ACTION

METHOD JobStart
VAR_INPUT
  aJobName       : T_MaxString;
  aJobGuid       : T_MaxString;
  nJobImageWidth : UDINT;
  nJobImageHeigth  : UDINT;
  nCamFrameWidth : UDINT;
  pGridSettings  : POINTER TO ST_DefGridSettings;
END_VAR
_bJobStartRequest := TRUE;
_nJobIdCtr := _nJobIdCtr + 1;
nPythonNewJob := _nJobIdCtr;

aPythonJobName := aJobName;
aPythonJobGuid := aJobGuid;
nPythonImageWidth := nJobImageWidth * GVL_Deformation.nC_GridSubReso;
nPythonImageHeight :=nJobImageHeigth * GVL_Deformation.nC_GridSubReso;
nPythonCamFrameWidth := nCamFrameWidth * GVL_Deformation.nC_GridSubReso;
IF pGridSettings <> 0 THEN
  nPythonImageOffsetY := pGridSettings^.nGridImageOffsetY * GVL_Deformation.nC_GridSubReso;
  nPythonGridPitchX := pGridSettings^.nGridPitchX * GVL_Deformation.nC_GridSubReso;
  nPythonGridPitchY := pGridSettings^.nGridPitchY * GVL_Deformation.nC_GridSubReso;
  nPythonGridSizeX := pGridSettings^.nGridSizeX * GVL_Deformation.nC_GridSubReso;
  nPythonGridSizeY := pGridSettings^.nGridSizeY * GVL_Deformation.nC_GridSubReso; 
END_IF
END_METHOD

METHOD JobStop : BOOL
VAR_INPUT
END_VAR
_bJobStopRequest:=TRUE;
END_METHOD

{attribute 'monitoring':='call'}
PROPERTY nErrorId : UDINT
GET
nErrorId := _nErrId;
END_GET
END_PROPERTY

(*
  Register CT to script.
  :return: TRUE if success.
*)
METHOD RegisterCT : BOOL
VAR_INPUT
  nCTIdx  : UDINT;  // ct memory index
END_VAR
IF NOT bScriptAlive THEN RETURN; END_IF  // script not ready, ignore request

nContainerToRegister := UDINT_TO_DINT(nCTIdx);
RegisterCT := TRUE;
END_METHOD

METHOD RemoveCT : BOOL
VAR_INPUT
    nCTID : UDINT;
END_VAR
IF NOT bScriptAlive THEN RETURN; END_IF  // script not ready, ignore request

nContainerToDelete := UDINT_TO_DINT(nCTID);

RemoveCT := TRUE;
END_METHOD

METHOD PRIVATE RunPythonScript : BOOL
VAR_INPUT
END_VAR
VAR
  ams_host : STRING;
  ams_port : UINT;
  cmd : STRING;
END_VAR
// config launcher cmd line for script
//   e.g. fBScriptLauncher.Start('172.17.7.143.1.1 851 PRG_PRINT.fbWorkerDefGrid_Python.fbPythonInterface --sim_mode');

// get parameter dynamically
ams_host := PRG_SYSTEMBASE.sO_AmsNetIdLocalHost;  // localhost
ams_port := TwinCAT_SystemInfoVarList._AppInfo.AdsPort;
cmd := F_Concat5(ams_host,' ',TO_STRING(ams_port),' ',sPythonInterfacePath);
fBScriptLauncher.sStartScriptName := 'start.bat';
fBScriptLauncher.sStopScriptName  := 'stop.bat';
fBScriptLauncher.Start(cmd);
END_METHOD

METHOD PRIVATE StopPythonScript
VAR_INPUT
END_VAR
fBScriptLauncher.Stop(nPID := THIS^.nPythonPID);
END_METHOD

{attribute 'monitoring':='call'}
PROPERTY tWatchdogTime : TIME
GET
tWatchdogTime := fbWatchdog.ET;
END_GET
END_PROPERTY

END_FUNCTION_BLOCK

// ---- POUs/Print/DefGrid/FB_GridDataExporter.TcPOU
(*Converts data to exportable formats*)
FUNCTION_BLOCK FB_GridDataExporter EXTENDS T_NamedBase
VAR_INPUT
  sOutputDir          : T_MaxString;    // output folder path (without \ at the end)
  sFileName           : T_MaxString;    // file name
  pFbImageDeformation : POINTER TO FB_ImageDeformation;
  nSelectGrid         : UDINT;          // 0=deformation calculated, 1=streamed grid
END_VAR
VAR_OUTPUT
  bBusy : BOOL;
END_VAR
VAR 
  // - file handling
  bSave, bLoad, bDump : BOOL;                   // commands
  fbSysFile           : FB_File_Basic_SysFile;  // config file access
  
  // - json handling
  fbJson              : FB_JsonSaxWriter;       // config writer (build json string from data)
  fbJsonRd            : FB_JsonDomParser;       // config parse on read/(edit) (parse json string into data)
  
  // - exported string
  sDoc                : STRING(nC_MaxStringSz); // big string holding all config file
  
  // helper
  sFileFormat         : STRING;        // selected file format 
  sOutputPath         : T_MaxString;   // file path to read/write
  bInitialized        : BOOL;
END_VAR
VAR CONSTANT
  nC_MaxStringSz      : UDINT := 10_000;
END_VAR

// self setup -----------------------------
// - init
IF NOT bInitialized THEN Init(); RETURN; END_IF

// check & fix parameter
IF pFbImageDeformation = 0 THEN RETURN; END_IF

   IF bDump THEN bDump := NOT DumpGrid(); 
ELSIF bSave THEN bSave := FileSave();
ELSIF bLoad THEN bLoad := FileLoad();
END_IF

bBusy := bSave OR bLoad OR bDump;

METHOD PRIVATE dumpCsv : BOOL
VAR_OUTPUT
  nSz : UDINT;
END_VAR
VAR
  i, k : UDINT := 0;
  nCamPoints : UDINT;
  sCamPoint : ST_CameraPointTbl;
  sGridPoint : ST_DeformationPointAccurate;
  nCols, nRows, nGridPoints : UDINT;
  sGridSettings : ST_DefGridSettings;
  tempStr : T_MaxString;
END_VAR
nCamPoints :=pFbImageDeformation^.nAvailableCamPoints;
nGridPoints := pFbImageDeformation^.nAvailableGridPoints;
sGridSettings := pFbImageDeformation^.sDefGridSettings;
nCols := sGridSettings.nGridSizeX;
nRows := sGridSettings.nGridSizeY;

// build export csv string ----------------------------------
// reset string
MEMSET(destAddr:=ADR(sDoc), fillByte:=0, n:=SIZEOF(sDoc));

// grid  (dx/dy)
//    col0    col1    col2
// |  0/0  |  1/0  |  2/0  | ...  |  row0
// |  0/1  |  1/1  |  2/1  | ...  |  row1
FOR i:=0 TO nRows-1 DO
  FOR k:=0 TO nCols-1 DO
    // get deformation point
    pFbImageDeformation^.getDeformationPoint(nCol:=k, nRow:=i, nSel:=nSelectGrid, sPoint=>sGridPoint, bWasSet=>);
    tempStr := F_Concat3(
      F_Concat2('dx:', TO_STRING(sGridPoint.dx)),
      F_Concat2('/dy:', TO_STRING(sGridPoint.dy)),
      F_Concat2(',', '')
    );
    CONCAT2(pSrcString1:=ADR(sDoc), pSrcString2:=ADR(tempStr), pDstString:=ADR(sDoc), nDstSize:=SIZEOF(sDoc));  // point dx/dy
  END_FOR
  tempStr := '$n';
  CONCAT2(pSrcString1:=ADR(sDoc), pSrcString2:=ADR(tempStr), pDstString:=ADR(sDoc), nDstSize:=SIZEOF(sDoc));  // newline
END_FOR

tempStr := '$n';
CONCAT2(pSrcString1:=ADR(sDoc), pSrcString2:=ADR(tempStr), pDstString:=ADR(sDoc), nDstSize:=SIZEOF(sDoc));

// cam
FOR k:=1 TO nCamPoints DO
  pFbImageDeformation^.getCamPointX(nIdx:=k, Pn=>sCamPoint);
  tempStr := F_Concat5(
    F_Concat2('x_ref:', TO_STRING(sCamPoint.sPoint.x_ref)), 
    F_Concat2('/y_ref:', TO_STRING(sCamPoint.sPoint.y_ref)), 
    F_Concat2('-dx:', TO_STRING(sCamPoint.sPoint.dx)), 
    F_Concat2('/dy:', TO_STRING(sCamPoint.sPoint.dy)),
    F_Concat2(',', '')
  );
  CONCAT2(pSrcString1:=ADR(sDoc), pSrcString2:=ADR(tempStr), pDstString:=ADR(sDoc), nDstSize:=SIZEOF(sDoc));
END_FOR

tempStr := '$n';
CONCAT2(pSrcString1:=ADR(sDoc), pSrcString2:=ADR(tempStr), pDstString:=ADR(sDoc), nDstSize:=SIZEOF(sDoc));

nSz := LEN2(pSTRING:=ADR(sDoc));
dumpCsv := TRUE;
END_METHOD

METHOD PRIVATE DumpGrid : BOOL 
VAR_OUTPUT
  nSz : UDINT;
END_VAR
IF    sFileFormat = 'csv'  THEN DumpGrid := dumpCsv(nSz=>nSz);
ELSE                            DumpGrid := dumpJson(nSz=>nSz);
END_IF
END_METHOD

METHOD PRIVATE dumpJson : BOOL
VAR_OUTPUT
  nSz : UDINT;
END_VAR
VAR
  i, k : UDINT := 0;
  nCamPoints : UDINT;
  sCamPoint : ST_CameraPointTbl;
  sGridPoint : ST_DeformationPointAccurate;
  nCols, nRows, nGridPoints : UDINT;
  sGridSettings : ST_DefGridSettings;
END_VAR
nCamPoints :=pFbImageDeformation^.nAvailableCamPoints;
nGridPoints := pFbImageDeformation^.nAvailableGridPoints;
sGridSettings := pFbImageDeformation^.sDefGridSettings;
nCols := sGridSettings.nGridSizeX;
nRows := sGridSettings.nGridSizeY;

// build big json string ----------------------------------
fbJson.ResetDocument();
fbJson.StartObject();
// {
    fbJson.AddKey(key:='Grid');
    fbJson.StartObject();
      fbJson.AddKey(key:='NumberOfGridPoints');
      fbJson.AddUdint(value:=nGridPoints);
      fbJson.AddKey(key:='GridPoints');
      fbJson.StartArray();
      FOR i:=1 TO nRows DO
        fbJson.StartArray();
        FOR k:=1 TO nCols DO
          fbJson.StartObject();
          pFbImageDeformation^.getDeformationPoint(nCol:=k-1, nRow:=i-1, nSel:=nSelectGrid, sPoint=>sGridPoint, bWasSet=>);
          fbJson.AddKey(key:='col');
          fbJson.AddDint(value:=sGridPoint.col);
          fbJson.AddKey(key:='row');
          fbJson.AddDint(value:=sGridPoint.row);
          fbJson.AddKey(key:='x_ref');
          fbJson.AddLreal(value:=sGridPoint.x_ref);
          fbJson.AddKey(key:='y_ref');
          fbJson.AddLreal(value:=sGridPoint.y_ref);
          fbJson.AddKey(key:='dx');
          fbJson.AddLreal(value:=sGridPoint.dx);
          fbJson.AddKey(key:='dy');
          fbJson.AddLreal(value:=sGridPoint.dy);
          fbJson.AddKey(key:='valid');
          fbJson.AddBool(value:=sGridPoint.valid);
          fbJson.EndObject();
        END_FOR
        fbJson.EndArray();
      END_FOR
      fbJson.EndArray();
    fbJson.EndObject();
    
    
    fbJson.AddKey(key:='Cam');
    fbJson.StartObject();
      fbJson.AddKey(key:='NumberOfCamPoints');
      fbJson.AddUdint(value:=nCamPoints);
      fbJson.AddKey(key:='CamPoints');
      fbJson.StartArray();
      FOR k:=1 TO nCamPoints DO
        pFbImageDeformation^.getCamPointX(nIdx:=k, Pn=>sCamPoint);
        fbJson.StartObject();
        fbJson.AddKey(key:='x_ref');
        fbJson.AddLreal(value:=sCamPoint.sPoint.x_ref);
        fbJson.AddKey(key:='y_ref');
        fbJson.AddLreal(value:=sCamPoint.sPoint.x_ref);
        fbJson.AddKey(key:='dx');
        fbJson.AddLreal(value:=sCamPoint.sPoint.dx);
        fbJson.AddKey(key:='dy');
        fbJson.AddLreal(value:=sCamPoint.sPoint.dy);
        fbJson.AddKey(key:='valid');
        fbJson.AddBool(value:=sCamPoint.sPoint.valid);
        fbJson.EndObject();
      END_FOR    
      fbJson.EndArray();
    fbJson.EndObject();
   
    // ]
fbJson.EndObject();
// '}'

fbJson.CopyDocument(sDoc, SIZEOF(sDoc));
// document is now in big string -----------------------------

nSz := LEN2(pSTRING:=ADR(sDoc));
dumpJson := TRUE;
END_METHOD

(*
  Load Simulation configuration file and apply settings / modes / config to each FB_Sim.
  :return: TRUE as long busy
*)
METHOD PRIVATE FileLoad : BOOL
VAR_OUTPUT
  nError : UDINT;
END_VAR
VAR_INST
  nState : UDINT := 0;
  eof : BOOL;
  sz : UDINT := 0;
  errCode : UDINT;
END_VAR
CASE nState OF
  0:  // idle
    LogLvl(Lvl:=E_LogSeverity.Detail, 'Load file');
    IF sOutputPath <> '' THEN
      sDoc := '';
      nState := nState + 1; // start immediately
    ELSE
      nState := 4;   // go to parse only
    END_IF
    errCode := 0;

    
  1:  // opening file
    IF NOT fbSysFile.Open(SName:=sOutputPath, eMode:=E_FileMode.rd, bBinary:=FALSE) THEN
      IF fbSysFile.nErrId <> 0 THEN 
        errCode := fbSysFile.nErrId;
        nState := 99;
      ELSE
			  nState := nState + 1;
      END_IF
		END_IF
    
  2:  // reading file
    IF NOT fbSysFile.Read(pStr:=ADR(sDoc), nSize:=SIZEOF(sDoc), nRdBytes=>sz, bEOF=>eof) THEN
      IF fbSysFile.nErrId <> 0 THEN 
        errCode := fbSysFile.nErrId;
        nState := 99;
      ELSIF NOT eof THEN
        LogError('File could not be loaded fully');
        nState := nState + 1;
      ELSE
			  nState := nState + 1;
      END_IF
		END_IF
    
  3:  // closing file
    LogLvl(Lvl:=E_LogSeverity.Debug, Msg:=F_Concat4('Loaded file, size=', TO_STRING(sz), ' file=', sOutputPath));
    IF NOT fbSysFile.Close() THEN
      IF fbSysFile.nErrId <> 0 THEN 
        errCode := fbSysFile.nErrId;
        nState := 99;
      ELSE
			  nState := nState + 1;
      END_IF
		END_IF
    
  4:  // parsing file
    //parseJson();
    nState := nState + 1;
    
  5:  // done
    nState := 0;
    
  99: // error
    LogError(F_Concat2('Load config stopped with error', TO_STRING(errCode)));
    nState := 0;
ELSE
  ;
END_CASE

// return values
nError := errCode;
FileLoad := nState <> 0;   // busy
END_METHOD

METHOD PRIVATE FileSave : BOOL
VAR_OUTPUT
  nError : UDINT;
END_VAR
VAR_INST
  nState : UDINT := 0;
  errCode : UDINT;
  nSz : UDINT;
END_VAR
CASE nState OF
  0:  // idle
    LogLvl(Lvl:=E_LogSeverity.Detail, Msg:=F_concat2('Saving file: ', sOutputPath));
    errCode := 0;
    nState := nState + 1;
      
  1:  // parsing file
    DumpGrid(nSz=>nSz);
    IF sOutputPath <> '' THEN
      nState := nState + 1;
    ELSE
      nState := 5;   // done (no file to write)
    END_IF
    
  2:  // opening file
    IF NOT   fbSysFile.Open(sName:=sOutputPath, eMode:=E_FileMode.wr, bBinary:=FALSE) THEN
      IF fbSysFile.nErrId <> 0 THEN 
        errCode := fbSysFile.nErrId;
        nState := 99;
      ELSE
			  nState := nState + 1;
      END_IF
		END_IF
    
  3:  // reading file
    IF NOT fbSysFile.Write(pStr:=ADR(sDoc), nSize:=nSz+1) THEN
      IF fbSysFile.nErrId <> 0 THEN 
        errCode := fbSysFile.nErrId;
        nState := 99;
      ELSE
			  nState := nState + 1;
      END_IF
		END_IF
    
  4:  // closing file
    LogLvl(Lvl:=E_LogSeverity.Debug, Msg:=F_Concat2('Saved file=', sOutputPath));
    IF NOT fbSysFile.Close() THEN
      IF fbSysFile.nErrId <> 0 THEN 
        errCode := fbSysFile.nErrId;
        nState := 99;
      ELSE
			  nState := nState + 1;
      END_IF
		END_IF
    
  5:  // done
    nState := 0;
    
  99: // error
    LogError(F_Concat2('Save file stopped with error', TO_STRING(errCode)));
    nState := 0;
ELSE
  ;
END_CASE

// return values
nError := errCode;
FileSave := nState <> 0;   // busy
END_METHOD

METHOD PRIVATE Init : BOOL
LogLevel := E_LogSeverity.Info;

Init:= bInitialized := TRUE;
END_METHOD

(*
  Parse json sting into data.
  :return: TRUE on success
*)
METHOD PRIVATE parseJson : BOOL
VAR
    // parser helper variables
  bHasMember  : BOOL;
  jsonRoot    : SJsonValue;   // full doc reference
  jsonModulAry, jsonIteratorModul, jsonIteratorEndModul, jsonModul : SJsonValue;  // handling module array
  jsonModeAry, jsonIteratorMode, jsonIteratorEndMode, jsonMode : SJsonValue;      // handling mode array
  jsonProp    : SJsonValue;   // effective single entry
  arySz       : UDINT;
  
  module      : T_MaxString;
  mode        : ST_SimModeDef;
  enable      : BOOL;
  active_mode : STRING;
END_VAR
// interpret new data ------------------------------
jsonRoot := fbJsonRd.ParseDocument(sJson:=jsonDoc);
bHasMember := fbJsonRd.HasMember(jsonRoot, 'modules');
IF (bHasMember) THEN
  // moules array
  bHasMember := FALSE;
  jsonModulAry := fbJsonRd.FindMember(jsonRoot, 'modules');
  arySz := fbJsonRd.GetArraySize(jsonModulAry);
  jsonIteratorModul := fbJsonRd.ArrayBegin(jsonModulAry);
  jsonIteratorEndModul := fbJsonRd.ArrayEnd(jsonModulAry);
  WHILE jsonIteratorModul <> jsonIteratorEndModul DO
    // for each module
    jsonModul := fbJsonRd.GetArrayValue(jsonIteratorModul);
    jsonProp := fbJsonRd.FindMember(jsonModul, 'module');
    module := fbJsonRd.GetString(jsonProp);   // simulation module name
    jsonProp := fbJsonRd.FindMember(jsonModul, 'sim_enable');
    enable := fbJsonRd.GetBool(jsonProp);   // simulation enable
    jsonProp := fbJsonRd.FindMember(jsonModul, 'active_mode');
    active_mode := fbJsonRd.GetString(jsonProp);   // simulation active mode
    // mode array
    jsonModeAry := fbJsonRd.FindMember(jsonModul, 'modes');
    arySz := fbJsonRd.GetArraySize(jsonModeAry);
    jsonIteratorMode := fbJsonRd.ArrayBegin(jsonModeAry);
    jsonIteratorEndMode := fbJsonRd.ArrayEnd(jsonModeAry);
    WHILE jsonIteratorMode <> jsonIteratorEndMode DO
      // for each mode
      jsonMode := fbJsonRd.GetArrayValue(jsonIteratorMode);
      mode.aMode := fbJsonRd.GetString(jsonIteratorMode);       // get mode name
      jsonProp := fbJsonRd.FindMember(jsonMode, mode.aMode);
      fbJsonrd.CopyJson(jsonProp, mode.sCfg, SIZEOF(mode.sCfg));    // get config data (raw json)
      
      // --- setup module ---
      setupSimModule(sModule:=module, sMode:=mode, enable:=enable, active_mode:=active_mode);
      // --------------------
      
      jsonIteratorMode := fbJsonRd.NextArray(jsonIteratorMode);
		END_WHILE
    // next modules
    jsonIteratorModul := fbJsonRd.NextArray(jsonIteratorModul);
  END_WHILE
END_IF

parseJson := TRUE;    // TODO: check for parsing errors
END_METHOD

METHOD startExport
VAR
  sFileEnding : STRING;
END_VAR
IF pFbImageDeformation = 0 THEN RETURN; END_IF

sFileEnding := F_FileGetExtension(aPath:=sFileName);
IF     sFileEnding = 'csv'  THEN sFileFormat := 'csv';
ELSIF  sFileEnding = 'json' THEN sFileFormat := 'json';  
END_IF

sOutputPath := F_Concat3(sOutputDir, '\', sFileName);

bSave := TRUE;
END_METHOD

END_FUNCTION_BLOCK

// ---- POUs/Print/DefGrid/FB_StartPositionDummy.TcPOU
(*
  A start position detection function block dummy.
  A dummy implementation to simulate start triggers at desired positions.
*)
FUNCTION_BLOCK FB_StartPositionDummy EXTENDS FB_BasePrint IMPLEMENTS I_StartPosDetect, I_PrintStatusClient, I_Sim
VAR_INPUT
  bTrigger                    : BOOL;       // manual trigger
  lPosition                   : DINT;       // current position [SubPx]
  fSpeed                      : LREAL;      // current speed [m/s]
  fResolution                 : LREAL;      // current print resolution [dpi*SubPx]
END_VAR

VAR
  // properties
  _bSim               : BOOL;       // simulatio mode active (PROPERTY)
  _bCreateTrigger     : BOOL;       // create new CT trigger (PROPERTY)
  _nStartPosX0        : DINT;       // create position for CT (absolut) [SubPx] (PROPERTY)
  _bAutoTrigger       : BOOL;       // automatic sheet triggers
  
  // config
  iJobDefinition      : CalmarCompPrint.I_JobDefinition;
  
  // local helper
  rfNewCT             : RF_TRIG;    // trigger new ct
  nSheetLength        : DINT;       // sheet length in [SubPx]
  nSheetGap           : DINT;       // sheet gap in [SubPx]
  nSheetEndPosition   : DINT;       // sheet end position [SubPx]
  nNextSheetPosition  : DINT;       // next trigger location
  fSheetPerHour       : LREAL;      // sheets per hour
  fSheetSpeed         : LREAL;      // [m/min] speed meter per minute
  tCheckTrigger       : TON;
  
  tCurrentTimeStamp   : T_DCTIME64; // get current timestamp
  fCurrentTimeStamp   : LREAL;      // current timestamp
  fSensorTimeStamp    : LREAL;      // sensor timestamp
  fDeltaDistance      : LREAL;      // distance that the substrate moved between the detection and the treatment of the information [m]
  
  rfTrig_Sim          : RF_TRIG;
END_VAR

VAR PERSISTENT
  // simulation configuration
  fSheetLength   : LREAL := 0.5;    // [m] sheet length (local or per job given)
  fSheetGap      : LREAL := 0.12;   // [m] gap between two sheets
END_VAR

// checks and fixes
IF iJobDefinition = 0 THEN RETURN; END_IF
IF fSpeed = 0 THEN RETURN; END_IF
IF fSheetLength = 0 THEN fSheetLength := 1; END_IF
IF fResolution = 0 THEN fResolution := 600*32; END_IF
rfTrig_Sim(CLK:=_bSim);
IF    rfTrig_Sim.RT THEN SimEnter(); 
ELSIF rfTrig_Sim.FT THEN SimExit(); END_IF

IF NOT _bSim THEN RETURN; END_IF

// calculations
fSheetSpeed := fSpeed * 60;  // [m/s] -> [m/min]
nSheetGap := F_MeterToSubPixel(fPosMeter := fSheetGap, fResoSubPx := fResolution);  // [m] -> [SubPx]
fSheetPerHour := (60*60)/((fSheetLength+fSheetGap)/fSpeed);
nSheetLength := F_MeterToSubPixel(fPosMeter := fSheetLength, fResoSubPx := fResolution);  // [mm] -> [SubPx]
nNextSheetPosition := _nStartPosX0 + nSheetLength + nSheetGap; 
tCheckTrigger(PT:=TO_TIME(((fSheetLength+fSheetGap)/fSpeed)*1000));

// internal trigger creation
IF (lPosition - nNextSheetPosition) > 0 AND _bAutoTrigger THEN
  bTrigger := TRUE;
  tCheckTrigger(IN:=FALSE);
  tCheckTrigger(IN:=TRUE);
END_IF

// on trigger
rfNewCT(CLK := bTrigger, RT => _bCreateTrigger);
IF _bCreateTrigger THEN   // new ct created
  bTrigger := FALSE;  // reset trigger
  
  (* Calculate the current and sensor time stamp (keep old code not really necessary because we use current timestamp)*)
  tCurrentTimeStamp := F_GetCurDcTaskTime64();
  fCurrentTimeStamp := (ULINT_TO_LREAL(tCurrentTimeStamp )) / 1_000_000.0; (*in ms*)
  fSensorTimeStamp  := fCurrentTimeStamp;
  fDeltaDistance := (fCurrentTimeStamp - fSensorTimeStamp) * 0.001 * fSpeed;  (*Distance that the substrate moved between the detection and the treatment of the information [m]*)
  
  // sheet start and sheet end pos in [SubPx]
  _nStartPosX0     := lPosition - F_MeterToSubPixel(fPosMeter := fDeltaDistance, fResoSubPx := fResolution);
  nSheetEndPosition := _nStartPosX0 + nSheetLength;
END_IF

{attribute 'monitoring' := 'call'}
(*Simulation is enabled set/get*)
PROPERTY bSimEnable : BOOL
GET
bSimEnable := _bSim;
END_GET
SET
_bSim := bSimEnable;
END_SET
END_PROPERTY

(*
  A new container detected.
  NOTE: a pulse only
*)
PROPERTY bStartTrig : BOOL
GET
bStartTrig := _bCreateTrigger;
END_GET
END_PROPERTY

(*
  A valid container detected.
*)
PROPERTY bValid : BOOL
GET
bValid := TRUE;
END_GET
END_PROPERTY

METHOD mJobPause
END_METHOD

METHOD mJobStart
VAR_INPUT
	sJobDef	: CalmarCompPrint.I_JobDefinition;
END_VAR
IF sJobDef = 0 THEN LogError('JobStart: no sJobDef given'); RETURN; END_IF

iJobDefinition := sJobDef;    // current job definition
fSheetLength := iJobDefinition.fSubstrateDepth;
END_METHOD

METHOD mJobStop
VAR_INPUT
	sStatus	: CalmarCompPrint.I_JobStatus;
END_VAR
iJobDefinition := 0;    // delete job definition
END_METHOD

METHOD mProduced
VAR_INPUT
	(* current progress*)
	sProgress	: CalmarCompPrint.I_JobProgress;
END_VAR
; // nothing to do
END_METHOD

(*
  Detected start position X0 (absolute) in [SubPx].
*)
PROPERTY nStartPositionX0 : DINT
GET
nStartPositionX0 := _nStartPosX0;
END_GET
END_PROPERTY

METHOD SimEnter : BOOL
LogInfo('Enter start position creator simulation');
_bSim := TRUE;

_nStartPosX0 := lPosition;
nSheetEndPosition := lPosition;
nNextSheetPosition := lPosition;
END_METHOD

METHOD SimExit : BOOL
LogInfo('Exit start position creator simulation');
_bSim := FALSE;
END_METHOD

END_FUNCTION_BLOCK

// ---- POUs/Print/DefGrid/FB_WorkerDefGrid_Delete.TcPOU
FUNCTION_BLOCK FB_WorkerDefGrid_Delete EXTENDS FB_WorkerDefGrid

METHOD PROTECTED  Attach : BOOL
VAR_INPUT
  iCT              : I_CT;                         (*container at triggered event position*)
END_VAR
IF SUPER^.Attach(iCT:=iCT) THEN

  // directyl release & delete the CT 
  Release(iCT:=_pAttachedCt^);

END_IF
END_METHOD

METHOD   mJobStart
VAR_INPUT
	sJobDef	: CalmarCompPrint.I_JobDefinition;
END_VAR
END_METHOD

METHOD  mJobStop
VAR_INPUT
	sStatus	: CalmarCompPrint.I_JobStatus;
END_VAR
END_METHOD

METHOD Release : BOOL
VAR_INPUT
  iCT              : I_CT;                         (*container at triggered event position*)
END_VAR
IF SUPER^.Release(iCT := iCT) THEN
  
  // it's the last worker so distroy attached CT
  IF _pCTM <> 0 THEN
    LogLvl(Lvl:=E_LogSeverity.Debug, Msg:=F_Concat2('DestroyCT: ', TO_STRING(iCT.pCT^.iId)));
    _pCTM^.DestroyCT(iCT:=iCT);
  END_IF
  
END_IF
END_METHOD

METHOD  work
SUPER^.work();

// release should already be done in attach
IF _pAttachedCt <> 0 THEN
  Release(iCT:=_pAttachedCt^);
END_IF
END_METHOD

END_FUNCTION_BLOCK

// ---- POUs/Print/DefGrid/FB_WorkerDefGrid_Inspection.TcPOU
FUNCTION_BLOCK FB_WorkerDefGrid_Inspection EXTENDS FB_WorkerDefGrid
VAR_INPUT
  EL2252_Feedback      AT%I* : BYTE := 16#FF;   (*(optional from version > EL2252-0000-0018) Output feedback bit coded, needs activation in PDO config of terminal
                                                      BIT 0: Output Kanal 1
                                                      BIT 1: Tristate Kanal 1
                                                      BIT 2: Output Kanal 2
                                                      BIT 3: Tristate Kanal 2*)
  nCurrentPosition           : DINT;            // current position in [SubPx]
  fCurrentSpeed              : LREAL;           // current speed in [m/s]
  fMaxMachineSpeed           : LREAL;           // max. machine speed in [m/s]
END_VAR
VAR_OUTPUT
  // IOs
  EL2252_Activate      AT%Q* : BYTE;            (*Oututs activation command (0->3 activate)*)
  EL2252_Output1       AT%Q* : BOOL;            (*Output1 bool state*)
  EL2252_StartTime     AT%Q* : T_DCTIME64;      (*Outputs activation timestamp*)
END_VAR
VAR
  // timestamp output  
  tNowDc                          : T_DCTIME64;       // Get Current Timestamp (now)
  fCycleTime : LREAL;            // Current calculated cycle time [s]
  
  // helper
  nDistBtwTriggerAndInspection_SubPx : DINT;   // worker position in [SubPx]
  nTriggerPos_SubPx : DINT;   // next trigger position [SubPx]
  tTriggerTime : T_DCTIME64;
  bTriggerActivating, bOutputActive : BOOL;
  bTriggerResetting, bResetActive : BOOL;     // output is currently set
  tResetTime : T_DCTIME64;
  nDelta_SubPx : DINT;
  bVerbose : BOOL;
END_VAR
VAR CONSTANT
  tC_CommTimeout : LREAL := 10.0/1000;   // 10ms in [s]
END_VAR

// nothing to do: see work() for cyclic call

METHOD PROTECTED  Attach : BOOL
VAR_INPUT
  iCT              : I_CT;                         (*container at triggered event position*)
END_VAR
VAR
  // temp pos
  deltaPosNowToTrigger_SubPx : DINT;
  deltaPosNowToTrigger_m : LREAL;
  // temp time
  deltaTime_s : LREAL;
  deltaTime_Dc : T_DCTIME64;
END_VAR
IF SUPER^.Attach(iCT:=iCT) THEN
  
  // calculate exact trigger position
  // X0 + WorkerInspection-Pos
  nTriggerPos_SubPx := iCT.GetPosX0(iTracker:=_iCTTracker) + nDistBtwTriggerAndInspection_SubPx;
  // delta to current pos
  deltaPosNowToTrigger_SubPx := nTriggerPos_SubPx - nCurrentPosition;  // delata position in [SubPx]
  deltaPosNowToTrigger_m := F_SubPixelToMeter(lPosSubPx:=deltaPosNowToTrigger_SubPx, fResSubPx:=_fPrintResolution*_fSubPxResolution);
  
  IF fCurrentSpeed = 0 THEN RETURN; END_IF   // crash avoid
  // delta in time
  deltaTime_s  := deltaPosNowToTrigger_m/fCurrentSpeed;
  IF bVerbose THEN LogInfo(F_Concat4('deltaTime', TO_STRING(deltaTime_s), ' deltaPosNowToTrigger_SubPx:', TO_STRING(deltaPosNowToTrigger_SubPx))); END_IF
  deltaTime_Dc := TO_ULINT(deltaTime_s * TO_LREAL(EC_DCTIME_TICKSPERSEC64));  
  
  // trigger time
  tTriggerTime := ULARGE_TO_ULINT(UInt64Add64(ULINT_TO_ULARGE(F_GetCurDcTaskTime64()), ULINT_TO_ULARGE(deltaTime_Dc)));  // TODO: apply the Output Timestamped compensation (analog to Input timestamp)
  setTrigger(bOut1:=TRUE, tTime:=tTriggerTime);
  bTriggerActivating := TRUE;
END_IF
END_METHOD

// cycle time in [s]
METHOD PRIVATE calcCycleTime : LREAL
VAR_INPUT
  tCurrent : T_DCTIME64;
END_VAR
VAR_INST
  tLastTimeStamp : T_DCTIME64 := 0;
END_VAR
calcCycleTime := (TO_LREAL(tCurrent) - TO_LREAL(tLastTimeStamp)) * 1E-9;
tLastTimeStamp  := tCurrent;  // memory timestamp
END_METHOD

METHOD   mJobStart
VAR_INPUT
	sJobDef	: I_JobDefinition;
END_VAR
END_METHOD

METHOD  mJobStop
VAR_INPUT
	sStatus	: I_JobStatus;
END_VAR
END_METHOD

METHOD Release : BOOL
VAR_INPUT
  iCT              : I_CT;                         (*container at triggered event position*)
END_VAR
IF SUPER^.Release(iCT := iCT) THEN
  ;  
END_IF
END_METHOD

METHOD PRIVATE resetOut
VAR
  tDistDc : T_DCTIME64;
  tULargeNow, tULargeDist : T_ULARGE_INTEGER;
END_VAR
// send FALSE in the next tC_CommTimeout
tDistDc := TO_ULINT(tC_CommTimeout * TO_LREAL(EC_DCTIME_TICKSPERSEC64));
tULargeNow := ULINT_TO_ULARGE(tNowDc);
tULargeDist := ULINT_TO_ULARGE(tDistDc);
tResetTime := ULARGE_TO_ULINT(UInt64Add64(tULargeNow, tULargeDist));
setTrigger(bOut1:=FALSE, tTime:=tResetTime);
END_METHOD

METHOD PRIVATE setTrigger
VAR_INPUT
  tTime : T_DCTIME64;
  bOut1 : BOOL;
END_VAR
EL2252_Activate  := 0;
EL2252_StartTime := tTime;
EL2252_Output1   := bOut1;
END_METHOD

METHOD  work
VAR
  bOutput1 : BOOL;
END_VAR
VAR_INST
  bTriggerActivating_mem : BOOL;
  bTriggerResetting_mem : BOOL;
  fPreAttachPos : LREAL;
END_VAR
// If you have issues with this block think about to implement a default EL2252_Activate output value
//   to sureley reset the output a next activation

SUPER^.work();

// Overwrite "default" tracking offset (Attach position)
fPreAttachPos := fMaxMachineSpeed * tC_CommTimeout;
_nTrackOffset := F_MeterToSubPixel(fPosMeter:=fPosition - fPreAttachPos, fResoSubPx:=_fPrintResolution*_fSubPxResolution);  // [pos domain] save position

// time & position updates
tNowDc     := F_GetCurDcTaskTime64();                         // current dc time (most accurate time stamp we have)
fCycleTime := calcCycleTime(tCurrent:=tNowDc);                // calculate cycle time of this fb
nDistBtwTriggerAndInspection_SubPx := F_MeterToSubPixel(fPosMeter:=fPosition, fResoSubPx:=_fPrintResolution*_fSubPxResolution);  // distance between Sensor and Inspectionin [SubPx] 

// output activation
IF bTriggerActivating AND bTriggerActivating_mem THEN  bTriggerActivating := FALSE;
  EL2252_Activate := 3;        // activate output config
  bOutputActive := TRUE;
END_IF
bTriggerActivating_mem := bTriggerActivating;

IF bOutputActive THEN
  // check if pos later than activation position --> reset
  nDelta_SubPx := F_MeterToSubPixel(fPosMeter:=tC_CommTimeout*fCurrentSpeed, fResoSubPx:=_fPrintResolution*_fSubPxResolution);
  IF ABS(nCurrentPosition - nTriggerPos_SubPx) > nDelta_SubPx THEN
    resetOut();
    bTriggerResetting := TRUE;
    bOutputActive := FALSE;
	END_IF
END_IF

IF bTriggerResetting AND bTriggerResetting_mem THEN  bTriggerResetting := FALSE;
  EL2252_Activate := 3;        // activate output config
  bResetActive := TRUE;
END_IF
bTriggerResetting_mem := bTriggerResetting;

IF bResetActive THEN
  // check if pos later than activation position --> reset
  IF UInt64Cmp64(ULINT_TO_ULARGE(tNowDc), ULINT_TO_ULARGE(tResetTime)) > 0 THEN
    bResetActive := FALSE;
	END_IF
END_IF

IF _pAttachedCt <> 0 THEN
  Release(iCT:=_pAttachedCt^);
END_IF
END_METHOD

END_FUNCTION_BLOCK

// ---- POUs/Print/DefGrid/FB_WorkerDefGrid_Print.TcPOU
FUNCTION_BLOCK FB_WorkerDefGrid_Print EXTENDS FB_WorkerDefGrid IMPLEMENTS I_PrintSubsystem
VAR_INPUT
  nEncoderPos           : DINT;   // Absolute virtual encoder
  bHardwareSync         : BOOL;
  bHardwareHold         : BOOL;
  {warning 'TODO: refactor according WorkerPrintWEU offsets in [m] and worker position without DetectToPrintDist?'}
  fPrintStartOffset     : LREAL;  // Offset from Module reference (configurative PU/PM/PG/PA ADS offset)
  fDetectOffset         : LREAL;  // StartDetect to Modoule reference
  fPrintYOffset         : LREAL;  // Y-Shift in ram memory
  fMasterSpeed          : LREAL;  // Speed [m/s]
  fPUElevation          : LREAL;  // PU distance from substrate [m]
  fPUPlate1_Temperature : LREAL;  // PU Plate1 temperature
  fPUPlate2_Temperature : LREAL;  // PU Plate2 temperature
END_VAR

VAR_OUTPUT
  bPrintActive          : BOOL;   // A print is activated / started
END_VAR

VAR
  // print
  // - references
  _pAdsPg            : POINTER TO FB_ADS_PG;      // pg ads reference (for pa)

  // grid specific
  // - references
  _iParamMediator    : I_ParamMediator;
    
  sDefGridSettings   : ST_DefGridSettings;  
  fCurrentColumnPos  : LREAL; // Currently column position
  fCurrentPreCharge  : LREAL; // Currently to be precharged
  nChargedColumns    : UDINT; // Already charged columns

  fbDropSpeedComp    : FB_DropSpeedComp;  
  bShowDropSpeedSetup: BOOL;

  fbPs               : FB_PS;
  fbPa               : FB_PA;
  fB_PcAdapter       : FB_PC_Adapter;

  _fPrintStartOffset : LREAL;   // internal print start offset (distance Cam -> PG1 + PG Offset + PU offset)
  _fWorkerOffset     : LREAL;   // worker offset from X0 static
  _nPosX0            : DINT;    // X0 for last attached CT (detected postion)
  _nPosXS            : DINT;    // XS for last attached CT (shifted print start position)
  _nPosXDelta        : DINT;    // Shift value X0 -> XS
  _fPosY             : LREAL;   // Y shift for last attached CT
  _fCurrentImgDepth  : LREAL;   // Job: current image length [m]
  _nPosDeltaToPrint  : DINT;    // delta pos in [SbuPx] from attach to print
  _bPaStarted        : BOOL;
  _bPaStartRequested : BOOL;
  fBStartTimeout     : TON;
  rTrigSync          : R_TRIG;
  _bForceDefGridOff  : BOOL;    // force deformation grid stream to ph off (send 0)
  _fPrintUnitWidth   : LREAL;   // print unit width [m]
  // grid settings
  _iPhGrid           : I_Correction_Grid;
  _sPhGridHwCfg      : ST_GridHwCfg;
    
  (*grid limit*)
  _fLimitCorrectionX : LREAL;     // correction limit in y (abs) [px]
  _fLimitCorrectionY : LREAL;     // correction limit in y (abs) [px]
  _bGridWasLimited   : BOOL;      // streamed grid was limited
    
  (*Messaging*)
  _bMsgInitialized   : BOOL;
  fb_MsgQueue        : FB_MSG_QUEUE;                        (*Message queue*)
  fb_MsgHandler      : FB_MSG_HANDLER;                      (*Message handler*)
  sL_MsgConfig       : ST_MSG_CONFIG;                       (*Message config*)
  fb_Msg             : ARRAY [1..iC_NUM_MSG] OF FB_MESSAGE; (*Messages*)
END_VAR

VAR PERSISTENT
  _fColumnsToPrecharge : LREAL := nC_COLUMNS_TO_PRECHARGE;
  _fStartShiftOffset   : LREAL := fC_START_SHIFT_OFFSET;
  _fStartShiftFactor   : LREAL := fC_START_SHIFT_FACTOR;
END_VAR

VAR CONSTANT
  iC_NUM_MSG               : UDINT := 5;
  nC_COLUMNS_TO_PRECHARGE  : LREAL := 2.1;
  fC_GRIDPOINT_STREAM_TIME : LREAL := 0.0025;     // time to stream one point [s]
  fC_START_SHIFT_FACTOR    : LREAL := -0.031;
  fC_START_SHIFT_OFFSET    : LREAL := -0.01;
END_VAR

IF NOT bInitialized THEN RETURN; END_IF

//TODO Add error/warnings
bError := FALSE;
nError := 0;

fbDropSpeedComp(fMasterSpeed:=fMasterSpeed, fDropTravelDistance:=fPUElevation);

//Start offset update
IF _fPrintStartOffset <> (fPrintStartOffset) THEN //Worker position changed
  IF _pAttachedCt = 0 THEN //Update only without attached container
    _fPrintStartOffset :=fPrintStartOffset;
	END_IF
END_IF

//Worker position update
IF _fWorkerPosition <> (_fPrintStartOffset + (_fStartShiftOffset + _fStartShiftFactor * fMasterSpeed)) THEN //Worker position changed (camera settings change)
  setupPosition();
END_IF

(*---- Messaging -----------------------*)
IF _bMsgInitialized THEN
  fb_MsgHandler();
  //fB_Msg[1](bI_Status := dfsdfdsf);
  fb_MsgQueue();
END_IF

PROPERTY aPaState : STRING
GET
aPaState := fbPa.aPaState;
END_GET
END_PROPERTY

METHOD PROTECTED  Attach : BOOL
VAR_INPUT
  iCT              : I_CT;                         (*container at triggered event position*)
END_VAR
Attach:=FALSE;

IF SUPER^.Attach(iCT:=iCT) THEN
  // Additional worker checks
    // - job is valid?
  IF _pAttachedCt^.pJob = 0 OR NOT _bJobActive THEN
    Release(iCT:=iCT);
    RETURN;   // do not print
  
  // CT valid & CT present
  ELSIF NOT _pAttachedCt^.bValid OR NOT _pAttachedCt^.bProductPresent THEN
    Release(iCT:=iCT);
    RETURN;   // do not print
  
  // Ignore start due to hardware hold  
  ELSIF bHardwareHold THEN
    _pNewAttached^.AbortDeformation(sReason:=EC_Print.ecPaAbortHold.Desc, Src:=_pEcSrc^, bHideLog:=TRUE);
    Release(iCT:=iCT);
    RETURN;   // do not print
  
  // - OK attach
  ELSE
    Attach := TRUE;
	END_IF
  
  
  //Prepare print station
  sDefGridSettings := _pAttachedCt^.sDefGridSettings;
  // fix some potential errors
  IF sDefGridSettings.nGridPitchX = 0 THEN sDefGridSettings.nGridPitchX :=1024; LogError(F_concat2('grid not configured, set default nGridPitchX=',TO_STRING(sDefGridSettings.nGridPitchX))); END_IF
  IF sDefGridSettings.nGridPitchY = 0 THEN sDefGridSettings.nGridPitchY :=1024; LogError(F_concat2('grid not configured, set default nGridPitchY=',TO_STRING(sDefGridSettings.nGridPitchY))); END_IF
  
  fbPs.bPrintEnable := iCT.bValid AND iCT.bProductPresent;
  fbPs.setGrid(sGrid:=sDefGridSettings);
  nChargedColumns := 0;

  //Start print, PA should be in READY or DONE
  
  // Set X print position
  _nPosX0 :=    _pAttachedCt^.nPosPrint_X0   {warning 'TODO: please write this in DMAX CreateCT CTM'}
              //- General Shift
              - F_MeterToSubPixel(fbDropSpeedComp.fDropPlacementError, _fPrintResolution*_fSubPxResolution); // - drop compensation*)
  _nPosXDelta := F_MeterToSubPixel(_fPrintStartOffset, _fPrintResolution*_fSubPxResolution); // + PG/PA Shift (additional PG offset 0 for firstLine)
  
  _nPosXS := _nPosX0 + _nPosXDelta;
  fB_PcAdapter.setPrintStartPos(nX0:=_nPosXS);
  
  // Set Y print position
  _fPosY := fPrintYOffset;
  fB_PcAdapter.setPrintYShift(nYShift:=FC_LREAL_TO_DINT(_fPosY));

  // check
  IF _nPosXS < nEncoderPos THEN
    LogWarning(Msg:=F_Concat4('Print start position:', TO_STRING(_nPosXS) ,' < Encoder position:', TO_STRING(nEncoderPos)));
	END_IF
  
  // save current distance to print position
  _nPosDeltaToPrint := _nPosXS - _iCTTracker.getPosAbs();   {warning 'TODO: to test if this matches after the change'}
  checkGridTiming();
  
  IF fbPa.printStart() THEN
    _bPaStarted := FALSE;
    _bPaStartRequested := TRUE;
    Attach:=TRUE;
    LogLvl(Lvl:=E_LogSeverity.Debug, F_Concat2('printStart:', _pAttachedCt^.print(0)));  // print container
    LogLvl(Lvl:=E_LogSeverity.Debug, F_Concat4('> XS:', TO_STRING(_nPosXS), ' = X0:', TO_STRING(_nPosX0)));
    LogLvl(Lvl:=E_LogSeverity.Debug, F_Concat4( 
                                         ' + shStartOffs:', TO_STRING(F_MeterToSubPixel(_fPrintStartOffset,_fPrintResolution*_fSubPxResolution)),
                                         ' - shDropComp:', TO_STRING(F_MeterToSubPixel(fbDropSpeedComp.fDropPlacementError,_fPrintResolution*_fSubPxResolution))
                                         ));
  ELSE  
    LogError(Msg:='PA not ready to start at attach');
    Release(iCT := iCT);
	END_IF
  
ELSE
  // parent attach failed case
END_IF
END_METHOD

PROPERTY bJobActive : BOOL
GET
bJobActive := _bJobActive;
END_GET
END_PROPERTY

PROPERTY bPausePrintCanEx : BOOL
GET
bPausePrintCanEx := FALSE; //Not implemented
END_GET
END_PROPERTY

PROPERTY bPcEnabled : BOOL
GET
bPcEnabled := fB_PcAdapter.bPcEnable;
END_GET
END_PROPERTY

PROPERTY bPrintEnabled : BOOL
GET
bPrintEnabled := _bEnable;
END_GET
END_PROPERTY

PROPERTY bPrinting : BOOL
GET
bPrinting := fbPa.bPrinting;
END_GET
END_PROPERTY

PROPERTY bPrintReady : BOOL
GET
bPrintReady := fbPa.bReady;
END_GET
END_PROPERTY

PROPERTY bQueueEmpty : BOOL
GET
bQueueEmpty := NOT fB_PcAdapter.bJobValid;
END_GET
END_PROPERTY

PROPERTY bStartPrintCanEx : BOOL
GET
bStartPrintCanEx := fbPa.bStartCanEx;
END_GET
END_PROPERTY

PROPERTY bStopPrintCanEx : BOOL
GET
bStopPrintCanEx := fbPa.bStopCanEx;
END_GET
END_PROPERTY

METHOD PRIVATE checkGridTiming : BOOL
VAR
END_VAR
// check for timing problems
IF fMasterSpeed <> 0 THEN

  // - check pre-charge at beginning
  IF _fColumnsToPrecharge * fC_GRIDPOINT_STREAM_TIME * _sPhGridHwCfg.nGridRoiRows >= F_SubPixelToMeter(lPosSubPx:=_nPosDeltaToPrint, fResSubPx:=_fPrintResolution*_fSubPxResolution) / fMasterSpeed  THEN
    LogError('Machine too fast for grid stream (for pre-charge at attach)');
  END_IF
  
 // - check charge time needed per columns vs machine speed and grid-sizeY
 IF fC_GRIDPOINT_STREAM_TIME * _sPhGridHwCfg.nGridRoiRows >= F_SubPixelToMeter(lPosSubPx:=TO_DINT(sDefGridSettings.nGridPitchX), fResSubPx:=_fPrintResolution) / fMasterSpeed THEN
   LogError('Machine too fast for grid stream (time rows per column)');
 END_IF

END_IF
END_METHOD

(*
  Limit correction to boundaries
  :return: TRUE if limited
*)
METHOD PRIVATE correctionLimit : BOOL
VAR_INPUT
  pPoint : POINTER TO ST_DeformationPointAccurate;
END_VAR
VAR
  bLimited : BOOL;
  nExeedX, nExeedY : LREAL;
END_VAR
// limit point correction to boundaries and inform
IF    pPoint^.dx >= _fLimitCorrectionX    THEN nExeedX := pPoint^.dx; pPoint^.dx := _fLimitCorrectionX;    bLimited:=TRUE; 
ELSIF pPoint^.dx <= -1*_fLimitCorrectionX THEN nExeedX := pPoint^.dx; pPoint^.dx := -1*_fLimitCorrectionX; bLimited:=TRUE;
ELSIF pPoint^.dy >= _fLimitCorrectionY    THEN nExeedY := pPoint^.dy; pPoint^.dy := _fLimitCorrectionY;    bLimited:=TRUE;
ELSIF pPoint^.dy <= -1*_fLimitCorrectionY THEN nExeedY := pPoint^.dy; pPoint^.dy := -1*_fLimitCorrectionY; bLimited:=TRUE;
END_IF
IF bLimited THEN 
  LogLvl(Lvl:=E_LogSeverity.Warning, Msg:=F_Concat5( 'Point=',TO_STRING(pPoint^.index),
                                                     F_Concat5(' c:r(',TO_STRING(pPoint^.col),'/',TO_STRING(pPoint^.row), ') '),
                                                     F_Concat4('dx:', TO_STRING(nExeedX), ' dy:', TO_STRING(nExeedY)),
                                                     ' correction exceeded limit')); 
END_IF

_bGridWasLimited := SEL(bLimited, FALSE, TRUE);
correctionLimit := bLimited;
END_METHOD

// current job image length in [m]
PROPERTY fImageLength : LREAL
GET
fImageLength := _fCurrentImgDepth;
END_GET
END_PROPERTY

PROPERTY fMaxPrintSpeed : LREAL
GET
fMaxPrintSpeed := 0;  // TODO: when i_pc_adapter has the info from pc/ph
END_GET
END_PROPERTY

(*
  Max. supported speed [m/s], 0 if not available
*)
{attribute 'monitoring':='call'}
PROPERTY fMaxSpeed : LREAL
GET
VAR
  nSpeedMpMin : DINT;
END_VAR
nSpeedMpMin := SEL(bWorkerEnable AND _pAdsPg <> 0, 0, _pAdsPg^.lMaxPrintSpeed);
fMaxSpeed := TO_LREAL(nSpeedMpMin)/60;
END_GET
END_PROPERTY

{attribute 'monitoring':='call'}
PROPERTY fStartShiftFactor : LREAL
GET
fStartShiftFactor := _fStartShiftFactor;
END_GET
SET
_fStartShiftFactor := fStartShiftFactor;
END_SET
END_PROPERTY

{attribute 'monitoring':='call'}
PROPERTY fStartShiftOffset : LREAL
GET
fStartShiftOffset := _fStartShiftOffset;
END_GET
SET
_fStartShiftOffset := fStartShiftOffset;
END_SET
END_PROPERTY

METHOD PROTECTED gridUpdate : BOOL
VAR_INPUT
  bEnableDeformation : BOOL;      // enable correction update, else correction (0/0) is written
  fPosRelToAttach : LREAL;        // position relative to attach of this worker
END_VAR
VAR
  sPoint : ST_DeformationPointAccurate;
  nRow : UDINT;
  bWasSet : BOOL;
  nAvailPoints : UDINT;
  nConvErr : UDINT;
END_VAR
VAR_INST
  nAvailPoints_mem : UDINT;
END_VAR
//TODO: rewrite this method to look cleaner (less if else)
gridUpdate:=TRUE;

// calculate grid column position
IF sDefGridSettings.nGridPitchX <> 0 THEN
  fCurrentColumnPos := fPosRelToAttach / (sDefGridSettings.nGridPitchX * _fSubPxResolution);   // calc grid column position relative to worker
END_IF

//Check for next correction update 
IF fCurrentColumnPos + _fColumnsToPrecharge > nChargedColumns AND nChargedColumns <= sDefGridSettings.nGridSizeX THEN
  IF bEnableDeformation THEN 
    // sync deformation points
    {warning 'TODO FIX: WHILE'}
    fCurrentPreCharge := fCurrentColumnPos + _fColumnsToPrecharge;
    WHILE FLOOR(fCurrentPreCharge) > nChargedColumns AND nChargedColumns <= sDefGridSettings.nGridSizeX DO
      nAvailPoints := _pAttachedCt^.nAvailableGridPoints;
      IF nAvailPoints >= sDefGridSettings.nGridSizeY * (nChargedColumns+1) THEN // Complete column available?
        nAvailPoints_mem := 0;
        LogLvl(Lvl:=E_LogSeverity.Debug, Msg:=F_Concat2('Charge CG col: ',TO_STRING(nChargedColumns)));
        FOR nRow := 0 TO sDefGridSettings.nGridSizeY - 1 DO
          // get points
          IF _pAttachedCt^.getDeformationPoint(nCol:=nChargedColumns, nRow:=nRow, nSel:=0, sPoint=>sPoint, bWasSet=>bWasSet) THEN
          
            IF NOT bWasSet THEN LogWarning(F_Concat5('Point[c(',TO_STRING(nChargedColumns),')/r(', TO_STRING(nRow),')] was not set')); END_IF  
                      
            // correction limitation
            correctionLimit(pPoint:=ADR(sPoint));
            
            // send point
            IF NOT fbPs.newGridPoint(sPoint:=sPoint) THEN
               LogError(Msg:='stream new point failed');
               gridUpdate:=FALSE;
               RETURN;
            END_IF
          ELSE
            LogError(Msg:='get new grid point failed');
            gridUpdate:=FALSE;
          END_IF
        END_FOR
        
        nChargedColumns := nChargedColumns + 1;
      ELSE
        IF nAvailPoints > nAvailPoints_mem THEN // log once or after every update of new available poinst
          LogError(Msg:='point column expected but not available');
        END_IF
        nAvailPoints_mem := nAvailPoints;
        gridUpdate:=FALSE;
        RETURN;
      END_IF 
    END_WHILE
  ELSE
    // send points with no deformation
      FOR nRow := 0 TO sDefGridSettings.nGridSizeY - 1 DO
        MEMSET(destAddr:=ADR(sPoint), fillByte:=0, n:=SIZEOF(sPoint));
        sPoint.col := TO_DINT(nChargedColumns);
        sPoint.row := TO_DINT(nRow);
        IF NOT fbPs.newGridPoint(sPoint:=sPoint) THEN
           LogError(Msg:='stream new point failed');
           gridUpdate:=FALSE;
           RETURN;
        END_IF
    END_FOR
    nChargedColumns := nChargedColumns + 1;
	END_IF
END_IF
END_METHOD

METHOD InitMsg : BOOL
VAR_INPUT
  pMsgInterface : POINTER TO ST_ADS_MSG_IF;
END_VAR
VAR
  nCtr : UDINT;
END_VAR
IF pMsgInterface = 0 THEN RETURN; END_IF

(*Messaging*)
sL_MsgConfig.bI_Enable       := TRUE;
sL_MsgConfig.pI_FbMsgHandler := ADR(fb_MsgHandler);
fb_MsgHandler.pI_MsgQueue    := ADR(fb_MsgQueue);
fb_MsgQueue.pI_MsgInterface  := pMsgInterface;
fb_MsgQueue.cI_MaxElement    := 6;

(*Messages*)
FOR nCtr := 1 TO iC_NUM_MSG DO
  fb_Msg[nCtr].pI_MsgConfig       := ADR(sL_MsgConfig);
  fb_Msg[nCtr].iI_MsgLocation     := 0;
END_FOR
//fb_Msg[1].iI_MsgNumber       := ;
// ...

_bMsgInitialized := TRUE;
END_METHOD

METHOD InitWorkerPrint : BOOL
VAR_INPUT
  pAdsPg                : POINTER TO FB_ADS_PG;       // pg ads reference (worker prints ads)
  iDefGridParamMediator : I_ParamMediator;
  fPrintUnitWidth       : LREAL;     // print unit width [m]
  fLimitCorrectionX     : LREAL;     // correction limit in y (abs) [px]
  fLimitCorrectionY     : LREAL;     // correction limit in y (abs) [px]
END_VAR
IF NOT bInitialized THEN LogError('Base Worker not initialized! call init() before'); RETURN; END_IF
IF pAdspg = 0 THEN LogError('InitWorkerPrint: invalid parameter proviced'); RETURN; END_IF
IF iDefGridParamMediator = 0 THEN bInitialized := FALSE; LogError('Invalid parameter, no valid param mediator'); RETURN; END_IF

// worker specific init
_pAdsPg := pAdsPg;
_iParamMediator := iDefGridParamMediator;

//Print Aggregate
_fPrintUnitWidth   := fPrintUnitWidth;
_fLimitCorrectionX := ABS(fLimitCorrectionX);
_fLimitCorrectionY := ABS(fLimitCorrectionY);

fbPa.bSyncAfterDone := FALSE;
fbPa.init(iPcAdapter := fB_PcAdapter, iPsInterface := fbPs);
END_METHOD

METHOD   mJobStart
VAR_INPUT
	sJobDef	: CalmarCompPrint.I_JobDefinition;
END_VAR
// Config workers static variables
_fCtSecurityReleasePos := F_MeterToSubPixel(fPosMeter:=(1.5 *sJobDef.fImageDepth) /1000, fResoSubPx:=_fPrintResolution*_fSubPxResolution);

IF NOT bWorkerEnable THEN RETURN; END_IF  // only if enabled

fbPa.jobStart(bEndless:=sJobDef.isEndless());

_bJobActive := TRUE;
_fCurrentImgDepth := sJobDef.fImageDepth/1000;

// grid settings update
IF _iPhGrid <> 0 THEN _sPhGridHwCfg := _iPhGrid.getGridHwCfg(); END_IF
END_METHOD

METHOD  mJobStop
VAR_INPUT
	sStatus	: CalmarCompPrint.I_JobStatus;
END_VAR
fbPa.jobStop();
_bJobActive := FALSE;
END_METHOD

PROPERTY pMsgConfig : POINTER TO ST_MSG_CONFIG
GET
pMsgConfig := ADR(sL_MsgConfig);
END_GET
END_PROPERTY

METHOD registerPc : BOOL
VAR_INPUT
  iNewPC : I_PC;
END_VAR
registerPc := fB_PcAdapter.registerPc(iNewPC := iNewPC);
END_METHOD

METHOD registerPh : BOOL
VAR_INPUT
  iPH : I_PH;
END_VAR
//Attach head to print station
IF iPH <> 0 THEN
  fbPs.registerPh(iNewPh:=iPH);
  _iPhGrid := iPH.iGridCorrection;
END_IF
END_METHOD

METHOD setupPosition
IF _pAttachedCt <> 0 THEN RETURN; END_IF    // Update only without attached container

// WorkerPosition =  PU<-CAM + CAM<-SheetDetect + StartShift calculated (with speed)
fPosition := _fPrintStartOffset + (_fStartShiftOffset + _fStartShiftFactor * fMasterSpeed);
END_METHOD

PROPERTY sPcFlags : CalmarCompPrint.ST_PC_FLAGS
GET
sPcFlags := fB_PcAdapter.sPcFlags;
END_GET
END_PROPERTY

PROPERTY sPcState :  CalmarCompPrint.ST_PG_STATUS
GET
VAR
  sJobStatus : ST_JobProgress;
END_VAR
sPcState.bStartPrintCanEx := fBPa.bStartCanEx;
sPcState.bStartPrintExec  := fBPa.bStartExec;
sPcState.bStopPrintCanEx  := fBPa.bStopCanEx;
sPcState.bStopPrintExec   := fBPa.bStopExec;
sPcState.bPausePrintCanEx := FALSE;       // obsolete ???
sPcState.bPausePrintExec  := FALSE;       // obsolete ???
sPcState.bReady           := fB_PcAdapter.bAllReady OR fB_PcAdapter.bAllDone;
sPcState.bError           := fB_PcAdapter.bError;
sPcState.bPrinting        := fB_PcAdapter.bAllPrinting;
sPcState.bLoad            := fB_PcAdapter.bAllPreparing;
sPcState.bArmed           := fB_PcAdapter.bAllPrinting OR fB_PcAdapter.bAllReady OR fB_PcAdapter.bAllDone OR fB_PcAdapter.bAllPreparing;
sPcState.bEnabled         := bWorkerEnable;
sPcState.bStartStrb       := fBPa.bStartStrb;
sPcState.bPcEnabled       := fB_PcAdapter.bPcEnable;
sPcState.lProductCount    := 0;            // obsolete ???
sPcState.sJobStatus       := sJobStatus;   // obsolete ???
END_GET
END_PROPERTY

METHOD  work
VAR
  bDeformErr : BOOL;
  nDeformStep : E_DeformationStep;
END_VAR
SUPER^.work();

(*Update virtual encoder on all controller boards*)
fB_PcAdapter.setEncoderPos(nEncoderPos);
fB_PcAdapter();

(*Call print aggregate*)
rTrigSync(CLK:=bHardwareSync); 
IF rTrigSync.Q THEN fbPa.sync(); END_IF   // external sync
fbPa.bHold := bHardwareHold;              // external hw hold
fbPa();

fBStartTimeout(IN := _bPaStartRequested,PT := T#60MS);

IF _pAttachedCt <> 0 AND bWorkerEnable THEN // Work only with attached container
  
  // check for generic error
  IF _pAttachedCt^.bValid AND bHardwareHold THEN
    // abort during printing
    _pNewAttached^.AbortDeformation(sReason:=EC_Print.ecPaAbortHold.Desc, Src:=_pEcSrc^, bHideLog:=TRUE);
  END_IF

  // Grid update
  bDeformErr := _pAttachedCt^.getDeformationStatus(eDStep=>nDeformStep);
  {warning 'TODO: re-enable gridUpdate()'}
(*
  IF NOT bDeformErr AND nDeformStep >= E_DeformationStep.gridStarted AND NOT _bForceDefGridOff THEN 
    IF NOT gridUpdate(bEnableDeformation:=TRUE) THEN
      _pAttachedCt^.AbortDeformation(sReason:='WorkerPrint: deformation point update failed', Src:=_pEcSrc^);
    END_IF
  ELSE
    // not started or error already --> erase deformation points
    gridUpdate(bEnableDeformation:=FALSE);
  END_IF  
*)  
  // PA control
  IF _bPaStartRequested THEN
    IF fbPa.bPrinting THEN
      _bPaStarted := TRUE;
      _bPaStartRequested := FALSE;
    ELSIF fBStartTimeout.Q THEN //Stop print at timeout to make ready for next container
      _bPaStarted := FALSE;
      _bPaStartRequested := FALSE;
      fbPa.printStop(bSyncedStop:=FALSE);
      _pNewAttached^.AbortDeformation(sReason:=EC_Print.ecPaStartErr.Desc, Src:=_pEcSrc^, bHideLog:=FALSE);
      Release(_pAttachedCt^);
		END_IF
  ELSIF _bPaStarted THEN
    //Release container when all points have been processed
    IF fbPa.bDone OR fbPa.bStop THEN
      _bPaStarted := FALSE;
      Release(_pAttachedCt^);
    (*ELSIF fbpa.bError THEN
      _pNewAttached^.AbortDeformation(sReason:=EC_Print.ecPaPrintErr.Desc, Src:=_pEcSrc^, bHideLog:=FALSE);
      Release(_pAttachedCt^);*)
    END_IF 
	END_IF
END_IF  

bPrintActive := _bPaStarted;

(*Logging config*)
fbPa.LogLevel := LogLevel;
fB_PcAdapter.LogLevel := LogLevel;
END_METHOD

END_FUNCTION_BLOCK

// ---- POUs/Print/DefGrid/FB_WorkerDefGrid_Python.TcPOU
{attribute 'reflection'} 
FUNCTION_BLOCK FB_WorkerDefGrid_Python EXTENDS FB_WorkerDefGrid IMPLEMENTS I_DeformationHandler
VAR_INPUT
END_VAR
VAR_OUTPUT
END_VAR
VAR
  // interface to py script
  fbPythonInterface : FB_PythonInterface;
  // references
  _iParamMediator : I_ParamMediator;
  
  // local copy of settings
  _bNewJob : BOOL;  // new job was activated
  _CamGridSettings : ST_CameraGridSettings;
  _DefGridSettings : ST_DefGridSettings;
  
  // local copy of job setting
  _aJobName         : T_MaxString;
  _aJobGuid         : T_MaxString;
  _fImageWidthM     : LREAL;          // image width in [m]
  _fImageDepthM     : LREAL;          // image depth in [m]
  

  // messages
  fbMsg_PythonNotRunning : FB_MESSAGE;
END_VAR

VAR CONSTANT
  fC_DEFAULT_WOKER_POSITION : LREAL := 0.01;      // default worker position in [m]
END_VAR

METHOD PROTECTED  Attach : BOOL
VAR_INPUT
  iCT              : I_CT;                         (*container at triggered event position*)
END_VAR
Attach := FALSE;
IF SUPER^.Attach(iCT:=iCT) THEN
  // OK, attached (enabled, was ok to be attached)
  IF _pNewAttached = 0 THEN RETURN; END_IF
  
  // setup check
  IF _iParamMediator = 0 THEN Release(iCT:=iCT); LogError('Invalid param mediator'); RETURN; END_IF
  
  // Additional worker checks
  // - do we have a valid job? used mode?
  IF _CamGridSettings.eCameraMode > E_CameraMode.NoCorrection AND (iCT.pJob = 0 OR NOT _bJobActive) THEN
    _pNewAttached^.AbortDeformation(sReason:='No valid job', Src:=_pEcSrc^, bHideLog:=FALSE);
     Release(iCT:=iCT);
     
  ELSIF _CamGridSettings.eCameraMode > E_CameraMode.NoCorrection THEN
    // OK attach
    // -- only create ct if a deformation is active
    IF CreateDefCt(iCT:=iCT) THEN
        // set state
        _pNewAttached^.StartScript(iDeformationHandler:=THIS^);
        // attached
        Attach := TRUE;
    END_IF
  ELSE
    ; // ignore attach
  END_IF
ELSE
  // parent attach failed
END_IF
END_METHOD

(*
  Create/Release virtual ct in deformation handlers.
  :return: TRUE if success
*)
METHOD PRIVATE CreateDefCt : BOOL;
VAR_INPUT
  iCT : I_CT;
END_VAR
IF iCT = 0 THEN RETURN; END_IF

IF _CamGridSettings.eCameraMode >= E_CameraMode.Live THEN
  IF fbPythonInterface.RegisterCT(iCT.pCT^.nMemIndex) THEN
    CreateDefCt := TRUE;
  ELSE
    _pAttachedCt^.AbortDeformation(sReason:='Could not register to script', Src:=_pEcSrc^, bHideLog:=FALSE);
  END_IF
ELSE
  CreateDefCt := TRUE;
END_IF
END_METHOD

METHOD DeleteCachedCt : BOOL
VAR_INPUT
	iCT	: I_CT;
END_VAR
DeleteDefCt(iCT:=iCT);
END_METHOD

(*
  Delete/Release virtual ct in deformation handlers.
  :return: TRUE if sucess
*)
METHOD DeleteDefCt : BOOL
VAR_INPUT
  iCT : I_CT;
END_VAR
IF iCT = 0 THEN RETURN; END_IF

IF _CamGridSettings.eCameraMode >= E_CameraMode.Live THEN
  IF fbPythonInterface.RemoveCT(iCT.pCT^.nMemIndex) THEN
    DeleteDefCt := TRUE;
  ELSE
    LogError('Could not delete ct in script');
  END_IF
END_IF
END_METHOD

